# B&R Automation Studio project KeePak_Bliss_Reworked
Automation Studio 4.7.7.74 SP; technology packages: Acp10Arnc0 5.8.2, mapp 1.71.0, TextSystem 

## Configuration MasterConfiguration_ServoRam

CPU X20CP0484, AutomationRuntime C4.72, Build 4.1.2, Safety 1.10, Vc V4.72.0

### Task classes (Cpu.sw)
```
Cyclic#1 (cycle 4000 us, tolerance 0 us):
  ModeContro <- ModeControl.ModeControl_ST.prg
  GluePattCt <- Recipes.GluePattCtrl.prg
Cyclic#2 (cycle 8000 us, tolerance 8000 us):
  AdhesiveCo <- Actuators.AdhesiveControl.prg
  FoldPushCo <- Actuators.FoldPushControl.prg
  VacuumCont <- Actuators.VacuumControl.prg [disabled]
  ServoRamHa <- ServoMotion.ServoRamHandler.prg
  ServoFeedH <- ServoMotion.ServoFeedHandler.prg
  MotionHand <- ServoMotion.MotionHandler.prg
  MappCalls <- ServoMotion.MappCalls.prg
  ServoPnPHa <- ServoMotion.ServoPnPHandler.prg
  BodyHopper <- ServoMotion.BodyHopperHandler.prg
  LeftHopper <- ServoMotion.LeftHopperHandler.prg
  RightHoppe <- ServoMotion.RightHopperHandler.prg
Cyclic#3 (cycle 48000 us, tolerance 48000 us):
  SafetySamp <- AsSafetySolution.SafetySample.prg
Cyclic#4 (cycle 100000 us, tolerance 100000 us):
  FlexTest1 <- Actuators.FlexTest.prg
Cyclic#7 (cycle 20000 us, tolerance 30000000 us):
  AlarmHandl <- AlarmControl.AlarmHandling.prg
Cyclic#8 (cycle 8000 us, tolerance 30000000 us):
  Recipes <- Recipes.Recipes.prg
  HMIControl <- HMI.HMIControl.prg
  FlexTest <- Actuators.NordsonComm.NordsonMBComm.prg
  NordsonExt <- Actuators.NordsonComm.NordsonExtendedComm.prg
  PatliteCom <- Stacklight.PatliteComm.prg
DataObjects: assl1, Acp10sys
NcDataObjects: acp10etxen <- ServoMotion.acp10etxen.dob, gBHop <- gFeedobj.gBHop.dob, gFeedi <- gFeedobj.gFeedi.dob, brake <- gFeedobj.brake.dob, disablebra <- gFeedobj.disablebrakecheck.dob
VcDataObjects: Visu <- HMI.Visu.dob, Panel <- AsSafetySolution.Panel.dob
Binaries: vccbtn, vcpdvnc, arialbd, vcmgr, vctcal, vcgclass, vcfile, vcctext, vccnum, TCData, vcpkat, udbdef, vcfntttf, arial, vccshape, vcalarm, vccpwd, vcdsloc, Visu01, vccdt, vccscale, vcchspot, vccbmp, vccstr, vcshared, vcrt, vcnet, Visu02, calibri, vcbclass, vcdsint, vcpdsw, vccovl, Visu03, vccddbox, vccpopup, Panel03, Panel02, vcchtml, Panel01, vcxml, vccurl, arsvcreg, TCLang, vcpfgen, vcclbox, Acp10map, acp10cfg, ServoFeed, ServoRam, sysconf, AlarmCfg, RcpCfg, Role, User, ashwd, iomap, arconfig, AlrmHstCfg, TC, asfw, ashwac, ServoPnP, BodyHop, LeftHop, RightHop, ServoHop, vcpdi815, vcptelo, vcpdihd, vcpk, vcpfppc7, vcpdi855, vcpfar00, TopLinMot, BotLinMot, RamCfg
Libraries: operator, runtime, astime, AsIecCon, standard, brsystem, sys_lib, Constants, Vacuum, FoldPush, GluePatt, SetRamPars, GrayToBin, AsBrStr, InvErrTxt, DistCalc, AsSafety, FileIO, AsXml, AsMbTcp, asstring, AsIOAcc, AsBrMath, Lib_PBFlx, AsEPL, DataObj, AsIODiag, Acp10man, Acp10par, NcGlobal, Acp10sdc, Acp10sim, Acp10_MC, MpAxis, MpBase, MpAlarmX, MpCom, MpRecipe, MappCall, Types, AxisFUBs, vcresman, areventlog, powerlnk
```

### Hardware
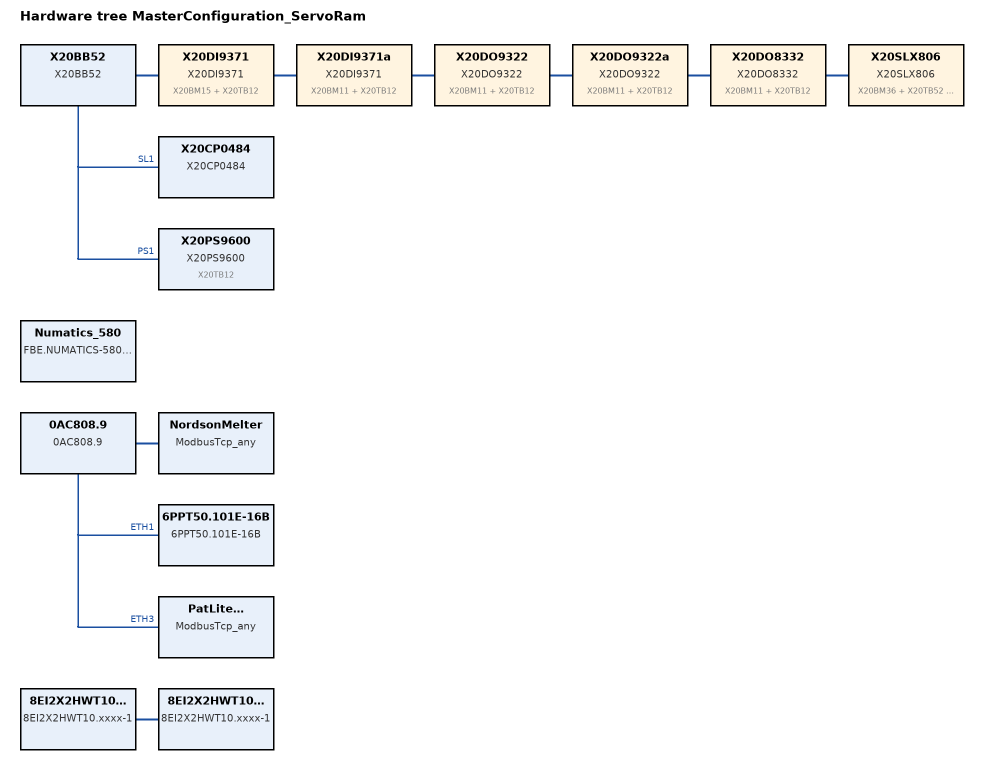
```
0AC808.9 : 0AC808.9 v1.0.0.0  [ETH1 -> 6PPT50.101E-16B.ETH1 [Cable Type=PowerlinkCable, Length=10, Version=1.0.0.2]; ETH2 -> NordsonMelter.ETH1 [Cable Type=PowerlinkCable, Length=10, Version=1.0.0.2]; ETH3 -> PatLite_LightStack.ETH1 [Cable Type=PowerlinkCable, Length=10, Version=1.0.0.2]]
6PPT50.101E-16B : 6PPT50.101E-16B v1.0.0.0  [ETH1 -> 0AC808.9.ETH1 [Cable Type=PowerlinkCable, Length=10, Version=1.0.0.2]; ETH2 -> X20CP0484.IF2 [Cable Type=PowerlinkCable, Length=10, Version=1.0.0.2]]
  Terminal = true
  Startmode = 1
  ShowBootlogoVNC = 1
  Mode = Manual
  InternetAddress = 192.168.0.222
  Subnetmask = 255.255.255.0
  ScreenRotation = 180
  SelectedFavoriteVNC = 192.168.0.100:5900
  Favorites_VNC1 = 192.168.0.100:5900  // Machine Display
  Favorites_VNC2 = 192.168.0.100:5901  // Safety Setup
  PasswordVNC = 2147
  LocalScaling = 1
  PasswordCIFS = 
  PasswordServiceEncrypt = 1
  PasswordServiceEncrypted = Sr1m/ubkTobKtMGmYG+OdX+pBVPXHNEV0toUjrnwIzvQUaZsN7HbgkMHcdX7NWbHkxunU2zcGZr9hHRCxdVEkcw0t0EkEZxQSM76MpE9s3WvBFtWwy/TiER4jA/5ccmygtG07vdCb9DlCJAeCcJdYe8VLadkZNOaNo2jGOliNnQ=
  VncKeyMappingFile = VC\6PPT30.101G-20B.dis
8EI2X2HWT10.xxxx-1 : 8EI2X2HWT10.xxxx-1 v2.2.0.1  [PLK2 -> 8EI2X2HWT10.xxxx-1a.PLK1 [Cable Type=PowerlinkCable, Length=10, Version=1.0.0.2]]
  MotionTP = Acp10Arnc0
  EnableDNA = on
  EPL_DNA_Head = 0
  EPL_DNA_Predecessor = 1
  Ax1Interface = Ax1EnDat
  Ax2Interface = Ax2EnDat
  Ax3Interface = Ax3EnDat
8EI2X2HWT10.xxxx-1a : 8EI2X2HWT10.xxxx-1 v2.2.0.1  [PLK1 -> 8EI2X2HWT10.xxxx-1.PLK2 [Cable Type=PowerlinkCable, Length=10, Version=1.0.0.2]; PLK2 -> X20CP0484.IF3 [Cable Type=PowerlinkCable, Length=10, Version=1.0.0.2]]
  MotionTP = Acp10Arnc0
  EnableDNA = on
  EPL_DNA_Head = 0
  EPL_DNA_HubPort = 1
  Ax1Interface = Ax1EnDat
  Ax2Interface = Ax2EnDat
  Ax3Interface = Ax3EnDat
NordsonMelter : ModbusTcp_any v1.0.6.0  [ETH1 -> 0AC808.9.ETH2 [Cable Type=PowerlinkCable, Length=10, Version=1.0.0.2]]
  IpAddress = 192.168.0.201
  UnitId = 1
Numatics_580 : FBE.NUMATICS-580-20150428-145500 v1.0 (OrderNumber=Numatics 580)
  Supervision = off
PatLite_LightStack : ModbusTcp_any v1.0.6.0 (Disabled=true)  [ETH1 -> 0AC808.9.ETH3 [Cable Type=PowerlinkCable, Length=10, Version=1.0.0.2]]
  Connector ETH2 (Disabled=true)
  IpAddress = 192.168.0.200
X20BB52 : X20BB52 v1.1.0.0
  Connector IF6:
    CycleTime = 2000
X20BM11 : X20BM11 v1.0.0.1  [X2X1 -> X20BM11b.X2X2]
X20BM11a : X20BM11 v1.0.0.1  [X2X1 -> X20BM15.X2X2]
X20BM11b : X20BM11 v1.0.0.1  [X2X1 -> X20BM11d.X2X2]
X20BM11d : X20BM11 v1.0.0.1  [X2X1 -> X20BM11a.X2X2]
X20BM15 : X20BM15 v1.0.1.0  [X2X1 -> X20BB52.IF6]
X20BM36 : X20BM36 v1.0.0.6  [X2X1 -> X20BM11.X2X2]
X20CP0484 : X20CP0484 v1.2.1.0  [SL -> X20BB52.SL1]
  Connector IF2:
    ActivateDevice = 1
    Mode = Manual
    InternetAddress = 192.168.0.100
    SubnetMask = 255.255.255.0
    InaNodeNumber = 0
    Vnc1
    VncVcObjectName1 = Visu
    VncKeyMappingFile1 = VC\PS2-Keyboard.dis
    VncAuthentication1 = 1
    VncPasswordViewOnly1 = 21472147
    VncPasswordViewControl1 = 2147
    VncMaxConnections1 = 4
    VncRefreshRate1 = 100
    Vnc2
    VncVcObjectName2 = Panel
    VncKeyMappingFile2 = VC\PS2-Keyboard1.dis
    VncAuthentication2 = 1
    VncPasswordViewOnly2 = 21472147
    VncPasswordViewControl2 = 2147
    VncPortNumber2 = 5901
    VncRefreshRate2 = 100
    ActivateModbus = 1
    NumSlaves = -1
    NumAllBlocks = -1
    MemSizeIn = -1
    MemSizeOut = -1
  Connector IF3:
    CycleTime = 4000
  ConfigurationID = KeePakVFDCaseErector_C70_10Inch
  UserPartitionSize = 100
  PermanentPvSize = 1024
  RemanentGlobalPvSize = 1024
  TimerDeviceType = EPLX2X
  TimerDevice = X20CP0484.IF3
  TaskClassIdleTime = 4000
  Cyclic1Duration = 4000
  Cyclic1Tolerance = 0
  Cyclic2Duration = 8000
  Cyclic2Tolerance = 8000
  Cyclic3Duration = 48000
  Cyclic3Tolerance = 48000
  Cyclic4Duration = 100000
  Cyclic4Tolerance = 100000
  Cyclic5Duration = 200000
  Cyclic5Tolerance = 200000
  Cyclic6Duration = 500000
  Cyclic6Tolerance = 500000
  Cyclic7Duration = 20000
  Cyclic7Tolerance = 30000000
  Cyclic8Duration = 8000
  Cyclic8Tolerance = 30000000
  FileDevice1
  FileDeviceName1 = recipes
  FileDevicePath1 = F:\
  EthernetDefaultGateway = 192.168.0.100
  FtpUser1
  FtpUsername1 = jeremy
  FtpUserPassword1 = CB9xa/tRkdxv0VtZFfoX4sbyc2/nOLcpzFFiUfDmX6w=
  FtpUserSalt1 = PVNzvqae
  FTPAccessRight1 = 0
X20DI9371 : X20DI9371 v1.0.2.0  [SS1 -> X20TB12.SS; SL -> X20BM15.SL1]
  Supervision = off
X20DI9371a : X20DI9371 v1.0.2.0  [SS1 -> X20TB12a.SS; SL -> X20BM11a.SL1]
X20DO8332 : X20DO8332 v1.0.2.0  [SS1 -> X20TB12e.SS; SL -> X20BM11.SL1]
  Supervision = off
  PowerSupply01 = on
X20DO9322 : X20DO9322 v1.0.3.0  [SS1 -> X20TB12d.SS; SL -> X20BM11d.SL1]
  Supervision = off
X20DO9322a : X20DO9322 v1.0.3.0  [SS1 -> X20TB12b.SS; SL -> X20BM11b.SL1]
X20PS9600 : X20PS9600 v1.0.1.0  [PS -> X20BB52.PS1; SS1 -> X20TB12f.SS]
X20SLX806 : X20SLX806 v1.10.5.0  [SS1 -> X20TB52.SS; SS2 -> X20TB52a.SS; SL -> X20BM36.SL1]
  Supervision = off
  SafeProject = SafeLOGIC-1
  SafeDesigner = 4.2.6.2
  DigitalOutput01 = viaSafeLOGIC
  DigitalOutput02 = viaSafeLOGIC
  DigitalOutput03 = viaSafeLOGIC
  DigitalOutput04 = viaSafeLOGIC
  DigitalOutput05 = viaSafeLOGIC
  DigitalOutput06 = viaSafeLOGIC
  UnsafeInputUINTs = 4
X20TB12 : X20TB12 v1.0.0.0
X20TB12a : X20TB12 v1.0.0.0
X20TB12b : X20TB12 v1.0.0.0
X20TB12d : X20TB12 v1.0.0.0
X20TB12e : X20TB12 v1.0.0.0
X20TB12f : X20TB12 v1.0.0.0
X20TB52 : X20TB52 v1.0.0.1
X20TB52a : X20TB52 v1.0.0.1
```

### Cpu.per - X20CP0484/Cpu.per
```iecst
VAR_CONFIG
	ServoFeed_EPD AT %M0; (* *)
	BodyHopper_EPD AT %M40; (* *)
	LeftHopper_EPD AT %M80; (* *)
	RightHopper_EPD AT %M120; (* *)
	ServoRam_EPD AT %M160; (* *)
	ServoPnP_EPD AT %M200; (* *)
	ServoRamFirstHomeExecuted AT %MX240; (* *)
	ServoFeedFirstHomeExecuted AT %MX241; (* *)
	BodyHopperFirstHomeExecuted AT %MX242; (* *)
	LeftHopperFirstHomeExecuted AT %MX243; (* *)
	RightHopperFirstHomeExecuted AT %MX244; (* *)
	ServoPnPFirstHomeExecuted AT %MX245; (* *)
	CycleCount AT %MD248; (* *)
	LubeCount AT %MD252; (* *)
END_VAR
```

### IoMap.iom - X20CP0484/IoMap.iom
```iecst
VAR_CONFIG
	Cyclic#1.::gIO.ModuleOKs[4] AT %IX."X20DO8332".ModuleOk;
	Cyclic#1.::gIO.DOs.GlueChannel1 AT %QX."X20DO8332".DigitalOutput01;
	Cyclic#1.::gIO.DOs.GlueChannel2 AT %QX."X20DO8332".DigitalOutput02;
	Cyclic#1.::gIO.DOs.GlueChannel3 AT %QX."X20DO8332".DigitalOutput03;
	Cyclic#1.::gIO.DOs.GlueChannel4 AT %QX."X20DO8332".DigitalOutput04;
	Cyclic#1.::gIO.DOs.ZeroEncoder AT %QX."X20DO8332".DigitalOutput08;
	Cyclic#1.::gIO.DOs.ResetSafety AT %QX."X20SLX806".BOOL101;
	Cyclic#1.::gIO.DIs.SafetyOK AT %IX."X20SLX806".BOOL001;
	Cyclic#1.::gIO.SafetyStatus.CabinetEStopStatus AT %IW."X20SLX806".UINT001;
	Cyclic#1.::gIO.SafetyStatus.SafetyProgramRunning AT %QX."X20SLX806".BOOL102;
	Cyclic#1.::gIO.SafetyStatus.SafetyProgramRunning AT %IX."X20SLX806".BOOL002;
	Cyclic#1.::gIO.ModuleOKs[6] AT %IX."X20SLX806".ModuleOk;
	Cyclic#1.::gIO.ModuleOKs[7] AT %IX."X20SC2212".ModuleOk;
	Cyclic#1.::gIO.SafetyStatus.GuardDoorsOK AT %IX."X20SLX806".BOOL003;
	Cyclic#1.::gIO.SafetyStatus.FrontEStopOK AT %IX."X20SLX806".BOOL004;
	Cyclic#1.::gIO.SafetyStatus.BackEstopOK AT %IX."X20SLX806".BOOL005;
	Cyclic#1.::gIO.DIs.AdhesivePhotoEye AT %IX."X20DI9371".DigitalInput01;
	Cyclic#1.::gIO.DIs.BodyDetect AT %IX."X20DI9371".DigitalInput04;
	Cyclic#1.::gIO.DIs.DownstreamSensorRaw AT %IX."X20DI9371".DigitalInput03;
	Cyclic#1.::gIO.DIs.BodyHopperLow AT %IX."X20DI9371".DigitalInput05;
	Cyclic#1.::gIO.DIs.AirPressureOK AT %IX."X20DI9371".DigitalInput02;
	::gIO.ModuleOKs[2] AT %IX."X20DI9371".ModuleOk;
	Cyclic#1.::gIO.DIs.BodyHopperMotor_OFF AT %IX."X20DI9371".DigitalInput09;
	Cyclic#1.::gIO.DIs.LeftHopperMotor_RUN AT %IX."X20DI9371".DigitalInput10;
	Cyclic#1.::gIO.DIs.LeftHopperMotor_OFF AT %IX."X20DI9371".DigitalInput11;
	Cyclic#1.::gIO.DIs.LeftHopperLow AT %IX."X20DI9371".DigitalInput06;
	Cyclic#1.::gIO.DIs.RightHopperLow AT %IX."X20DI9371".DigitalInput07;
	Cyclic#1.::gIO.DIs.BodyHopperMotor_RUN AT %IX."X20DI9371".DigitalInput08;
	Cyclic#1.::gIO.DIs.RightHopperMotor_RUN AT %IX."X20DI9371".DigitalInput12;
	Cyclic#1.::gIO.DOs.FoldingHoldVacuum AT %QX."X20DO9322".DigitalOutput03;
	Cyclic#1.::gIO.DOs.BodyVacuumOn AT %QX."X20DO9322".DigitalOutput01;
	Cyclic#1.::gIO.DOs.SidePanelHoldVacuum AT %QX."X20DO9322".DigitalOutput02;
	Cyclic#1.::gIO.DOs.PushOn AT %QX."X20DO9322".DigitalOutput04; (*24 VDC / 0.5 A, source **Normally the Pushers go here***)
	Cyclic#1.::gIO.DOs.AmberLightStack AT %QX."X20DO9322".DigitalOutput05;
	Cyclic#1.::gIO.DOs.GreenLightStack AT %QX."X20DO9322".DigitalOutput06;
	Cyclic#1.::gIO.DOs.RedLightStack AT %QX."X20DO9322".DigitalOutput07;
	Cyclic#1.::gIO.DOs.AirOn AT %QX."X20DO9322".DigitalOutput08;
	Cyclic#1.::gIO.DOs.Pneumatics580ControlWord1 AT %QW."Numatics_580".Out01_I3201Out;
	Cyclic#1.::gIO.ModuleOKs[7] AT %IX."Numatics_580".ModuleOk;
	Cyclic#1.::gIO.DIs.Pneumatics580StatusWord3 AT %IW."Numatics_580".In03_I3403;
	::b_ModuleStatus AT %IX."NordsonMelter".ModuleOk;
	Cyclic#1.::gIO.DIs.RightHopperMotor_OFF AT %IX."X20DI9371a".DigitalInput01;
	Cyclic#1.::gIO.DIs.BodyVacuumAchieved AT %IX."X20DI9371a".DigitalInput02;
	Cyclic#1.::gIO.DIs.SidePickVacuumAchieved AT %IX."X20DI9371a".DigitalInput03;
	Cyclic#1.::gIO.DIs.SideFoldVacuumAchieved AT %IX."X20DI9371a".DigitalInput04;
	Cyclic#1.::gIO.DOs.OutConveyorOn_1 AT %QX."X20DO9322".DigitalOutput09;
	Cyclic#1.::gIO.DOs.OutConveyorOn_2 AT %QX."X20DO9322".DigitalOutput10;
	Cyclic#1.::gIO.DOs.OutConveyorOn_3 AT %QX."X20DO9322".DigitalOutput11;
	Cyclic#1.::gIO.DOs.SidePickCylinder AT %QX."X20DO9322a".DigitalOutput01;
	Cyclic#1.::gIO.DOs.RightSideFoldCylinder AT %QX."X20DO9322a".DigitalOutput04;
	Cyclic#1.::gIO.DOs.LeftSideFoldCylinder AT %QX."X20DO9322a".DigitalOutput03;
	Cyclic#1.::gIO.DOs.CompressionCylinder AT %QX."X20DO9322a".DigitalOutput05;
	Cyclic#1.::gIO.DOs.BodyKicker AT %QX."X20DO9322".DigitalOutput12;
	Cyclic#1.::GuideCylinder AT %QX."X20DO9322a".DigitalOutput02;
	Cyclic#1.::gIO.DIs.LubricationCounter AT %IX."X20DI9371a".DigitalInput05;
	Cyclic#1.::gIO.DIs.BodyPickHome AT %IX."X20DI9371a".DigitalInput06;
END_VAR
```

### LeftHop.mpaxisbasic - X20CP0484/Motion/LeftHop.mpaxisbasic
```
Element mpLeftHopper (Type=mpaxisbasic)
  AxisConfiguration:
    Axis:
      MeasurementUnit = 1
  Alarms = MpAlarmX
    mapp.AlarmX.Core.Configuration:
      [0]:
        Severity = 110
      [1]:
        Severity = 110
      [2]:
        Severity = 110
      [3]:
        Severity = 110
      [4]:
        Severity = 110
      [5]:
        Severity = 110
      [6]:
        Severity = 110
      [7]:
        Severity = 110
      [8]:
        Severity = 110
      [9]:
        Severity = 110
      [10]:
        Severity = 110
      [11]:
        Severity = 110
      [12]:
        Severity = 110
      [13]:
        Severity = 110
      [14]:
        Severity = 110
      [15]:
        Severity = 110
```

- Safety project (password-protected, skipped)

## Logical view

### Global.var
```iecst
VAR RETAIN
	BodyHopperFirstHomeExecuted : BOOL;
	BodyHopper_EPD : MC_ENDLESS_POSITION;
END_VAR
VAR
	b_ModuleStatus : BOOL;
END_VAR
VAR RETAIN
	CycleCount : UDINT;
END_VAR
VAR
	DistanceAfterLatch : REAL;
	FeedInCycle : BOOL;
	FeedPosFinal : LREAL;
	FeedPositionCapture : LREAL;
	FeedServoBusy : BOOL;
	gActivePage : USINT;
	gAdhesiveCtrlInterface : AdhesiveCtrlInterface_typ;
	gAirPressureAlarmActive : BOOL;
	gAlarmActive : BOOL;
	gAlarmSystemActive : BOOL;
	gAutoTune : BOOL;
	gBodyHopper : ACP10AXIS_typ;
	gBodyHopperInterface : Axis_Interface_typ;
	gBotLinAxis : ACP10AXIS_typ;
	gBotLinAxis_1 : ACP10AXIS_typ;
	gChangePage : USINT;
	gCurrentLimitHit : BOOL;
	gCyclesToFinish : SINT;
	gDownstreamBlocked : BOOL;
END_VAR
VAR RETAIN
	gEndlessPosBot : MC_ENDLESS_POSITION;
	gEndlessPosTop : MC_ENDLESS_POSITION;
END_VAR
VAR
	gFoldPushCtrlInterface : FoldPushCtrlInterface_typ := (Parameters:=(LinMotBotFolder:=(Parameter:=(MpBasicParameters:=(Home:=(Mode:=mpAXIS_HOME_MODE_RESTORE_POS,Position:=0,StartVelocity:=25,HomingVelocity:=5,Acceleration:=500,StartDirection:=mpAXIS_HOME_DIR_NEGATIVE,TorqueLimit:=0.5,BlockDetectionPositionError:=4,PositionErrorStopLimit:=10),Jog:=(Velocity:=2)))),LinMotTopFolder:=(Parameter:=(MpBasicParameters:=(Home:=(Mode:=mpAXIS_HOME_MODE_RESTORE_POS,Position:=0,StartVelocity:=25,HomingVelocity:=5,Acceleration:=500,StartDirection:=mpAXIS_HOME_DIR_NEGATIVE,TorqueLimit:=0.5,BlockDetectionPositionError:=4,PositionErrorStopLimit:=10),Jog:=(Velocity:=2))))));
	gForceBodyKicker : BOOL;
	gHighSeverityAlarmActive : BOOL;
	gHMI : HMIControl_typ;
	gHomingParameters : Home_Parameters_typ;
	gIO : IO_typ;
	gIsSimulated : BOOL;
	gLeftHopper : ACP10AXIS_typ;
	gLeftHopperInterface : Axis_Interface_typ;
	gLowSeverityAlarmActive : BOOL;
	gModeControlInterface : ModeCtrlInterface_typ;
	gNumActiveAlarms : UDINT;
	gNumAlarms : UDINT;
	gOffDelayCompensation : REAL;
	gOnDelayCompensation : REAL;
END_VAR
VAR CONSTANT
	gPassword : ARRAY[0..2] OF STRING[80] := ['','0911','6866'];
END_VAR
VAR
	gPnPAtStopPosition : BOOL;
	gPusherOn : BOOL;
	gRamAtStopPosition : BOOL;
	gRamCtrlInterface : RamControlInterface_typ;
	gRamWaitingOnBox : BOOL;
END_VAR
VAR RETAIN
	gRecipeInterface : {REDUND_UNREPLICABLE} RecipeCtrlInterface_typ := (0);
END_VAR
VAR
	gRightHopper : ACP10AXIS_typ;
	gRightHopperInterface : Axis_Interface_typ;
	gSafetyNotOKAlarmActive : BOOL;
	gServoFeed : ACP10AXIS_typ;
	gServoFeedInterface : Axis_Interface_typ;
	gServoFeed_1 : ACP10AXIS_typ;
	gServoPnP : ACP10AXIS_typ;
	gServoPnPInterface : Axis_Interface_typ;
	gServoRam : ACP10AXIS_typ;
	gServoRamInterface : Axis_Interface_typ;
	gServoRam_1 : ACP10AXIS_typ;
	gSoftwareReset : BOOL;
	gTopLinAxis : ACP10AXIS_typ;
	gTopLinAxis_1 : ACP10AXIS_typ;
	GuideCylinder : BOOL;
	gUserLevel : USINT;
	gVacCtrlInterface : VacCtrlInterface_typ;
	HoperLowStop : BOOL;
	HopperLowTime : TIME := T#7s;
	InfeedBoxPresent : BOOL;
END_VAR
VAR RETAIN
	LeftHopperFirstHomeExecuted : BOOL;
	LeftHopper_EPD : MC_ENDLESS_POSITION;
	LubeCount : UDINT;
END_VAR
VAR
	LubricationOK : BOOL;
	Melter : DUT_NDSN_Flex;
	PhotoEyeSeen : BOOL;
END_VAR
VAR RETAIN
	RightHopperFirstHomeExecuted : BOOL;
	RightHopper_EPD : MC_ENDLESS_POSITION;
	ServoFeedFirstHomeExecuted : BOOL;
	ServoFeed_EPD : MC_ENDLESS_POSITION;
END_VAR
VAR
	ServoPnPAutoHome : BOOL;
END_VAR
VAR RETAIN
	ServoPnPFirstHomeExecuted : BOOL;
	ServoPnP_EPD : MC_ENDLESS_POSITION;
END_VAR
VAR
	ServoRamAutoHome : BOOL;
	ServoRamBusy : BOOL;
	ServoRamClear : BOOL;
END_VAR
VAR RETAIN
	ServoRamFirstHomeExecuted : BOOL;
END_VAR
VAR
	ServoRamTrigger : BOOL;
END_VAR
VAR RETAIN
	ServoRam_EPD : MC_ENDLESS_POSITION;
END_VAR
VAR
	StopFeed : BOOL;
END_VAR
```

### Program Logical/Actuators/AdhesiveControl

#### Init.st
```iecst
PROGRAM _INIT
	(* Insert code here *)
	gAdhesiveCtrlInterface.Parameters.NumAdhesiveChannels := 4;

	DistanceAfterLatch := 1500; //make this large so that the machine doesn't start dispensing glue before it ever sees a photo eye. This will reset to 0 and count up once the photo eye is seen

END_PROGRAM
```

### Program Logical/Actuators/NordsonComm/NordsonMBComm

#### MbApp.typ
```iecst
(********************************************************************
 * COPYRIGHT -- Bernecker + Rainer
 ********************************************************************
 * Program: MbApp
 * File: MbApp.typ
 * Author: Bernecker + Rainer
 * Created: October 22, 2009
 ********************************************************************
 * Local data types of program MbApp
 ********************************************************************)

TYPE
	ModbusTCP_Handling_States_enum :
		(
		MB_IDLE := 0,
		MB_REQUEST_SET_TEMPS2,
		MB_REQUEST_SET_TEMPS,
		MB_READ_SET_TEMPS2,
		MB_READ_SET_TEMPS,
		MB_REQUEST_ACT_TEMPS2,
		MB_REQUEST_ACT_TEMPS,
		MB_READ_ACT_TEMPS2,
		MB_READ_ACT_TEMPS,
		MB_REQUEST_MELTER_STATUS,
		MB_READ_MELTER_STATUS,
		MB_REQUEST_ADH_USE,
		MB_READ_ADH_USE,
		MB_WRITE_REGISTERS,
		MB_READ_REGISTERS,
		MB_REQUEST_MACHINE_STATUS,
		MB_WRITE_SET_TEMP2,
		MB_WRITE_SET_TEMP,
		MB_VERIFY_SET_TEMP_WRITE2,
		MB_VERIFY_SET_TEMP_WRITE,
		MB_REQUEST_ATS_ALARMS,
		MB_READ_ATS_ALARMS,
		MB_ERROR := 999
		);
END_TYPE
```

#### MbApp.var
```iecst
(********************************************************************
 * COPYRIGHT -- Bernecker + Rainer
 ********************************************************************
 * Program: MbApp
 * File: MbApp.var
 * Author: Bernecker + Rainer
 * Created: October 22, 2009
 ********************************************************************
 * Local variables of program MbApp
 ********************************************************************)
VAR
	state : ModbusTCP_Handling_States_enum;
	mb_station : STRING[50];
	write_register_address : UINT;
	num_registers_to_write : UINT;
	read_register_address : UINT;
	num_registers_to_read : UINT;
	ReadMultipleRegisters : mbReadHoldingRegisters;
	WriteMultipleRegisters : mbWriteMultipleRegisters;
	MBError : UINT;
	testIdx : USINT;
	DummyPacket2 : NordsonRxPacket_typ;
	DummyPacket : NordsonRxPacket_typ;
	NordsonRxPacket : NordsonRxPacket_typ;
	testChannel : USINT;
	NordsonTxPacket : NordsonTxPacket_typ;
	FeedbackCycleTimer : TON;
	MelterCmd : USINT;
	TempChannelToWrite : USINT;
	StandbyTimer : TON;
	FirstTimeCopySetTemps : BOOL;
END_VAR
```

#### MbApp.st
```iecst
(********************************************************************
 * COPYRIGHT -- Bernecker + Rainer
 ********************************************************************
 * Program: MbApp
 * File: MbApp.st
 * Author: Bernecker + Rainer
 * Created: October 22, 2009
 ********************************************************************
 * Implementation of program MbApp
 * State Nomenclature: "request" is a write to the nordson melter asking for some data
 * 					   "read" is a read from the nordson melter of the previously requested data
 *                     "write" is a write to the nordson melter asking to write some data to the melter
 *                     "verify" is a read from the nordson melter where we check to see that the write was accepted
 ********************************************************************)

PROGRAM _INIT

	NordsonTxPacket.Byte0_MelterControl := 16#1;
	NordsonTxPacket.Byte1_Command := 3;
	NordsonTxPacket.Byte2_Data_Index := 16#78;
	NordsonTxPacket.Byte3_Channel_Num := 16#3;
	NordsonTxPacket.Byte4_5_WriteData := 0;
	NordsonTxPacket.Byte6_7_Mot1Spd := 0;
	NordsonTxPacket.Byte8_9_Mot2Spd := 0;
	NordsonTxPacket.Byte10_11_Mot3Spd := 0;
	NordsonTxPacket.Byte12_13_Mot4Spd := 0;
	NordsonTxPacket.Byte14_15_NotUsed := 0;

	state := MB_IDLE;

	(* init values *)
	mb_station 			:= 'IF2.ST2';					(* path to modbus station *)
	write_register_address	:= 1024;						(* register address on modbus station *)
	read_register_address	:= 0;						(* register address on modbus station *)
	num_registers_to_write := 8;
	num_registers_to_read := 8;

	testChannel := CHANNEL_ACT_TEMP_START;
	testIdx := IDX_ACT_TEMP;

	gAdhesiveCtrlInterface.Commands.MelterOn := TRUE;
	gAdhesiveCtrlInterface.Commands.PumpsOn := TRUE;
	//gAdhesiveCtrlInterface.Parameters.NordsonComms.StandbyTimeoutTime := T#2h;
	//Removed Standby due to Waco machine going into Standby at random times. Added 05/15/2024

	FirstTimeCopySetTemps := FALSE;

END_PROGRAM

PROGRAM _CYCLIC

	IF(gAdhesiveCtrlInterface.Parameters.FeedbackIsModbusTCP) THEN
		gHMI.StatusDatapoints.NordsonModbusSDP := UNHIDE + UNLOCK;
	ELSE
		gHMI.StatusDatapoints.NordsonModbusSDP := HIDE + LOCK;
	END_IF

	//StandbyTimer.IN := NOT(gRamCtrlInterface.Status.Running) AND NOT(gAdhesiveCtrlInterface.Commands.MelterStandbyOn);
	StandbyTimer.IN := NOT(gServoRamInterface.Status.InMotion OR gServoPnPInterface.Status.InMotion OR gServoFeedInterface.Status.InMotion OR
							gBodyHopperInterface.Status.InMotion OR gLeftHopperInterface.Status.InMotion OR gRightHopperInterface.Status.InMotion)
						AND NOT(gAdhesiveCtrlInterface.Commands.MelterStandbyOn);

	StandbyTimer.PT := gAdhesiveCtrlInterface.Parameters.NordsonComms.StandbyTimeoutTime;
	StandbyTimer();

	IF(StandbyTimer.Q) THEN
		gAdhesiveCtrlInterface.Commands.MelterStandbyOn := TRUE;
	END_IF

	//clearing standby on command shiuld turn standby off. Changed standbyoff to True
	IF(gAdhesiveCtrlInterface.Commands.MelterStandbyOff) THEN
		gAdhesiveCtrlInterface.Commands.MelterStandbyOff := TRUE;
		gAdhesiveCtrlInterface.Commands.MelterStandbyOn := FALSE;
	END_IF

	IF((gAdhesiveCtrlInterface.Status.NordsonInStandby) AND (gAdhesiveCtrlInterface.Parameters.FeedbackIsModbusTCP)) THEN
		gHMI.StatusDatapoints.NordsonStandbyOffSDP := UNHIDE + UNLOCK;
	ELSE
		gHMI.StatusDatapoints.NordsonStandbyOffSDP := HIDE + LOCK;
	END_IF

	//if nordson feedback is bypassed, the error count should reset to 0
	IF gAdhesiveCtrlInterface.Parameters.NordsonComms.ByPassFeedback THEN
		gAdhesiveCtrlInterface.Parameters.NordsonComms.ConsecutiveErrorCount := 0;
	END_IF

	CASE state OF

		MB_IDLE:
			FeedbackCycleTimer.IN := ((gAdhesiveCtrlInterface.Parameters.FeedbackIsModbusTCP) AND (gAdhesiveCtrlInterface.Parameters.NordsonComms.ByPassFeedback = FALSE));

			IF(gAdhesiveCtrlInterface.Parameters.FeedbackIsModbusTCP = FALSE) THEN
				gAdhesiveCtrlInterface.Parameters.NordsonComms.ConsecutiveErrorCount := 0;
			END_IF

			IF(gAdhesiveCtrlInterface.Commands.WriteChannelTemp) THEN
				gAdhesiveCtrlInterface.Commands.WriteChannelTemp := FALSE;
				IF gAdhesiveCtrlInterface.Parameters.NordsonComms.GlobalSetTemp <> 0 THEN
					gAdhesiveCtrlInterface.Parameters.NordsonComms.ChannelSetTempRequested[0] := gAdhesiveCtrlInterface.Parameters.NordsonComms.GlobalSetTemp;
					gAdhesiveCtrlInterface.Parameters.NordsonComms.ChannelSetTempRequested[1] := gAdhesiveCtrlInterface.Parameters.NordsonComms.GlobalSetTemp;
					gAdhesiveCtrlInterface.Parameters.NordsonComms.ChannelSetTempRequested[2] := gAdhesiveCtrlInterface.Parameters.NordsonComms.GlobalSetTemp;
					gAdhesiveCtrlInterface.Parameters.NordsonComms.ChannelSetTempRequested[3] := gAdhesiveCtrlInterface.Parameters.NordsonComms.GlobalSetTemp;
					gAdhesiveCtrlInterface.Parameters.NordsonComms.ChannelSetTempRequested[4] := gAdhesiveCtrlInterface.Parameters.NordsonComms.GlobalSetTemp;
					gAdhesiveCtrlInterface.Parameters.NordsonComms.ChannelSetTempRequested[5] := gAdhesiveCtrlInterface.Parameters.NordsonComms.GlobalSetTemp;
					gAdhesiveCtrlInterface.Parameters.NordsonComms.ChannelSetTempRequested[6] := gAdhesiveCtrlInterface.Parameters.NordsonComms.GlobalSetTemp;
					gAdhesiveCtrlInterface.Parameters.NordsonComms.ChannelSetTempRequested[7] := gAdhesiveCtrlInterface.Parameters.NordsonComms.GlobalSetTemp;
					gAdhesiveCtrlInterface.Parameters.NordsonComms.ChannelSetTempRequested[8] := gAdhesiveCtrlInterface.Parameters.NordsonComms.GlobalSetTemp;
					gAdhesiveCtrlInterface.Parameters.NordsonComms.ChannelSetTempRequested[9] := gAdhesiveCtrlInterface.Parameters.NordsonComms.GlobalSetTemp;
					gAdhesiveCtrlInterface.Parameters.NordsonComms.GlobalSetTemp := 0;
				END_IF
				TempChannelToWrite := 0;
				state := MB_WRITE_SET_TEMP;

			ELSIF(FeedbackCycleTimer.Q) THEN
				FeedbackCycleTimer.IN := FALSE;
				state := MB_REQUEST_MELTER_STATUS;
			END_IF

		MB_REQUEST_MELTER_STATUS:

			WriteMultipleRegisters.enable := 1;
			NordsonTxPacket.Byte0_MelterControl := MelterCmd;
			NordsonTxPacket.Byte1_Command := READ_COMMAND;
			NordsonTxPacket.Byte2_Data_Index := IDX_MELTER_STATUS;
			NordsonTxPacket.Byte3_Channel_Num := 0;

			IF((WriteMultipleRegisters.status = ERR_FUB_ENABLE_FALSE) OR (WriteMultipleRegisters.status = ERR_FUB_BUSY)) THEN
				//do nothing
			ELSIF(WriteMultipleRegisters.status = ERR_OK) THEN
				WriteMultipleRegisters.enable := 0;
				state := MB_READ_MELTER_STATUS;
			ELSE
				WriteMultipleRegisters.enable := 0;
				MBError := WriteMultipleRegisters.status;
				state := MB_ERROR;
			END_IF

		MB_READ_MELTER_STATUS:

			ReadMultipleRegisters.enable := 1;

			IF((ReadMultipleRegisters.status = ERR_FUB_ENABLE_FALSE) OR (ReadMultipleRegisters.status = ERR_FUB_BUSY)) THEN
				//do nothing
			ELSIF(ReadMultipleRegisters.status = ERR_OK) THEN

				ReadMultipleRegisters.enable := 0;

				IF(NordsonRxPacket.Byte2_Ack_Data_Index = NordsonTxPacket.Byte2_Data_Index) THEN

					gAdhesiveCtrlInterface.Parameters.NordsonComms.MelterStatus := NordsonRxPacket.Byte4_5_Read_Data_0;
					gAdhesiveCtrlInterface.Parameters.NordsonComms.MelterIsOn := (gAdhesiveCtrlInterface.Parameters.NordsonComms.MelterStatus <> 8); //melter status == 8 => melter is not on

					DecodeStatus;

					//the melter MUST see a 0 for its ON command before it sees a 1. Send a 0 if the unit is faulted OR we have previously told it to turn on. and it never came on
				//	IF((gAdhesiveCtrlInterface.Parameters.NordsonComms.UnitFaulted) OR ((gAdhesiveCtrlInterface.Parameters.NordsonComms.MelterIsOn = FALSE) AND (NordsonTxPacket.Byte0_MelterControl.0 = TRUE))) THEN
					IF((gAdhesiveCtrlInterface.Parameters.NordsonComms.MelterIsOn = FALSE) AND (NordsonTxPacket.Byte0_MelterControl.0 = TRUE)) THEN
						MelterCmd := MELTER_OFF + PUMPS_OFF; //melter off, pumps off
					ELSE

						MelterCmd := 0;
						IF(gAdhesiveCtrlInterface.Commands.MelterOn) THEN
							MelterCmd := MelterCmd + MELTER_ON;
						END_IF

						IF((gAdhesiveCtrlInterface.Commands.PumpsOn) AND (gAdhesiveCtrlInterface.Status.UnitReady)) THEN
							MelterCmd := MelterCmd + PUMPS_ON; //only turn the pump on if the melter is ready
						END_IF

						IF((gAdhesiveCtrlInterface.Commands.MelterStandbyOn = FALSE) OR ((gAdhesiveCtrlInterface.Status.NordsonInStandby = FALSE) AND NordsonTxPacket.Byte0_MelterControl.6 = TRUE)) THEN
							//do not standby on
						ELSIF (gAdhesiveCtrlInterface.Commands.MelterStandbyOn = TRUE) THEN
							MelterCmd := MelterCmd + STANDBY_ON; //only turn the pump on if the melter is ready
						END_IF
					END_IF

					state := MB_REQUEST_SET_TEMPS;
				ELSE
					//stay in this state and re-execute read
				END_IF

			ELSE
				ReadMultipleRegisters.enable := 0;
				MBError := ReadMultipleRegisters.status;
				state := MB_ERROR;
			END_IF

		MB_REQUEST_SET_TEMPS:

			WriteMultipleRegisters.enable := 1;
			NordsonTxPacket.Byte0_MelterControl := MelterCmd;
			NordsonTxPacket.Byte1_Command := READ_COMMAND;
			NordsonTxPacket.Byte2_Data_Index := IDX_SET_TEMP;
			NordsonTxPacket.Byte3_Channel_Num := CHANNEL_SET_TEMP_START;

			IF((WriteMultipleRegisters.status = ERR_FUB_ENABLE_FALSE) OR (WriteMultipleRegisters.status = ERR_FUB_BUSY)) THEN
				//do nothing
			ELSIF(WriteMultipleRegisters.status = ERR_OK) THEN
				WriteMultipleRegisters.enable := 0;
				gAdhesiveCtrlInterface.Parameters.NordsonComms.ConsecutiveErrorCount := 0;
				state := MB_READ_SET_TEMPS;
			ELSE
				WriteMultipleRegisters.enable := 0;
				MBError := WriteMultipleRegisters.status;
				state := MB_ERROR;
			END_IF

		MB_READ_SET_TEMPS:

			ReadMultipleRegisters.enable := 1;

			IF((ReadMultipleRegisters.status = ERR_FUB_ENABLE_FALSE) OR (ReadMultipleRegisters.status = ERR_FUB_BUSY)) THEN
				//do nothing
			ELSIF(ReadMultipleRegisters.status = ERR_OK) THEN
				ReadMultipleRegisters.enable := 0;
				gAdhesiveCtrlInterface.Parameters.NordsonComms.ConsecutiveErrorCount := 0;

				IF((NordsonRxPacket.Byte2_Ack_Data_Index = NordsonTxPacket.Byte2_Data_Index) AND
					(NordsonRxPacket.Byte3_Ack_Channel_Num = NordsonTxPacket.Byte3_Channel_Num)) THEN

					DecodeStatus;

					gAdhesiveCtrlInterface.Parameters.NordsonComms.ChannelSetTempActual[0] := NordsonRxPacket.Byte4_5_Read_Data_0;
					gAdhesiveCtrlInterface.Parameters.NordsonComms.ChannelSetTempActual[1] := NordsonRxPacket.Byte6_7_Read_Data_1;
					gAdhesiveCtrlInterface.Parameters.NordsonComms.ChannelSetTempActual[2] := NordsonRxPacket.Byte8_9_Read_Data_2;
					gAdhesiveCtrlInterface.Parameters.NordsonComms.ChannelSetTempActual[3] := NordsonRxPacket.Byte10_11_Read_Data_3;
					gAdhesiveCtrlInterface.Parameters.NordsonComms.ChannelSetTempActual[4] := NordsonRxPacket.Byte12_13_Read_Data_4;
                    gAdhesiveCtrlInterface.Parameters.NordsonComms.ChannelSetTempActual[5] := NordsonRxPacket.Byte14_15_Read_Data_5;

					IF (FirstTimeCopySetTemps = FALSE) THEN
						gAdhesiveCtrlInterface.Parameters.NordsonComms.ChannelSetTempRequested := gAdhesiveCtrlInterface.Parameters.NordsonComms.ChannelSetTempActual;
						FirstTimeCopySetTemps := TRUE;
					END_IF

					state := MB_REQUEST_SET_TEMPS2; //for now, just go back to idle. Future versions need to read more stuff
				ELSE
					//stay in this state and re-execute read
				END_IF
			ELSE
				ReadMultipleRegisters.enable := 0;
				MBError := ReadMultipleRegisters.status;
				state := MB_ERROR;
			END_IF

		MB_REQUEST_SET_TEMPS2:

			WriteMultipleRegisters.enable := 1;
			NordsonTxPacket.Byte0_MelterControl := MelterCmd;
			NordsonTxPacket.Byte1_Command := READ_COMMAND;
			NordsonTxPacket.Byte2_Data_Index := IDX_SET_TEMP;
			NordsonTxPacket.Byte3_Channel_Num := 7;

			IF((WriteMultipleRegisters.status = ERR_FUB_ENABLE_FALSE) OR (WriteMultipleRegisters.status = ERR_FUB_BUSY)) THEN
				//do nothing
			ELSIF(WriteMultipleRegisters.status = ERR_OK) THEN
				WriteMultipleRegisters.enable := 0;
				gAdhesiveCtrlInterface.Parameters.NordsonComms.ConsecutiveErrorCount := 0;
				state := MB_READ_SET_TEMPS2;
			ELSE
				WriteMultipleRegisters.enable := 0;
				MBError := WriteMultipleRegisters.status;
				state := MB_ERROR;
			END_IF

		MB_READ_SET_TEMPS2:

			ReadMultipleRegisters.enable := 1;

			IF((ReadMultipleRegisters.status = ERR_FUB_ENABLE_FALSE) OR (ReadMultipleRegisters.status = ERR_FUB_BUSY)) THEN
				//do nothing
			ELSIF(ReadMultipleRegisters.status = ERR_OK) THEN
				ReadMultipleRegisters.enable := 0;
				gAdhesiveCtrlInterface.Parameters.NordsonComms.ConsecutiveErrorCount := 0;

				IF((NordsonRxPacket.Byte2_Ack_Data_Index = NordsonTxPacket.Byte2_Data_Index) AND
					(NordsonRxPacket.Byte3_Ack_Channel_Num = NordsonTxPacket.Byte3_Channel_Num)) THEN

					DecodeStatus;

					gAdhesiveCtrlInterface.Parameters.NordsonComms.ChannelSetTempActual[6] := NordsonRxPacket.Byte4_5_Read_Data_0;
					gAdhesiveCtrlInterface.Parameters.NordsonComms.ChannelSetTempActual[7] := NordsonRxPacket.Byte6_7_Read_Data_1;
					gAdhesiveCtrlInterface.Parameters.NordsonComms.ChannelSetTempActual[8] := NordsonRxPacket.Byte8_9_Read_Data_2;
					gAdhesiveCtrlInterface.Parameters.NordsonComms.ChannelSetTempActual[9] := NordsonRxPacket.Byte10_11_Read_Data_3;

					IF (FirstTimeCopySetTemps = FALSE) THEN
						gAdhesiveCtrlInterface.Parameters.NordsonComms.ChannelSetTempRequested := gAdhesiveCtrlInterface.Parameters.NordsonComms.ChannelSetTempActual;
						FirstTimeCopySetTemps := TRUE;
					END_IF

					state := MB_REQUEST_ACT_TEMPS; //for now, just go back to idle. Future versions need to read more stuff
				ELSE
					//stay in this state and re-execute read
				END_IF
			ELSE
				ReadMultipleRegisters.enable := 0;
				MBError := ReadMultipleRegisters.status;
				state := MB_ERROR;
			END_IF

		MB_REQUEST_ACT_TEMPS:

			WriteMultipleRegisters.enable := 1;
			NordsonTxPacket.Byte0_MelterControl := MelterCmd;
			NordsonTxPacket.Byte1_Command := READ_COMMAND;
			NordsonTxPacket.Byte2_Data_Index := IDX_ACT_TEMP;
			NordsonTxPacket.Byte3_Channel_Num := CHANNEL_ACT_TEMP_START;

			IF((WriteMultipleRegisters.status = ERR_FUB_ENABLE_FALSE) OR (WriteMultipleRegisters.status = ERR_FUB_BUSY)) THEN
				//do nothing
			ELSIF(WriteMultipleRegisters.status = ERR_OK) THEN
				WriteMultipleRegisters.enable := 0;
				state := MB_READ_ACT_TEMPS;
			ELSE
				WriteMultipleRegisters.enable := 0;
				MBError := WriteMultipleRegisters.status;
				state := MB_ERROR;
			END_IF

		MB_READ_ACT_TEMPS:

			ReadMultipleRegisters.enable := 1;

			IF((ReadMultipleRegisters.status = ERR_FUB_ENABLE_FALSE) OR (ReadMultipleRegisters.status = ERR_FUB_BUSY)) THEN
				//do nothing
			ELSIF(ReadMultipleRegisters.status = ERR_OK) THEN
				ReadMultipleRegisters.enable := 0;

				IF((NordsonRxPacket.Byte2_Ack_Data_Index = NordsonTxPacket.Byte2_Data_Index) AND
					(NordsonRxPacket.Byte3_Ack_Channel_Num = NordsonTxPacket.Byte3_Channel_Num)) THEN

					DecodeStatus;

					DummyPacket := NordsonRxPacket;

					gAdhesiveCtrlInterface.Parameters.NordsonComms.ChannelActTemp[0] := NordsonRxPacket.Byte4_5_Read_Data_0;
					gAdhesiveCtrlInterface.Parameters.NordsonComms.ChannelActTemp[1] := NordsonRxPacket.Byte6_7_Read_Data_1;
					gAdhesiveCtrlInterface.Parameters.NordsonComms.ChannelActTemp[2] := NordsonRxPacket.Byte8_9_Read_Data_2;
					gAdhesiveCtrlInterface.Parameters.NordsonComms.ChannelActTemp[3] := NordsonRxPacket.Byte10_11_Read_Data_3;
					gAdhesiveCtrlInterface.Parameters.NordsonComms.ChannelActTemp[4] := NordsonRxPacket.Byte12_13_Read_Data_4;
                    gAdhesiveCtrlInterface.Parameters.NordsonComms.ChannelActTemp[5] := NordsonRxPacket.Byte14_15_Read_Data_5;

					state := MB_REQUEST_ACT_TEMPS2;
				ELSE
					//stay in this state and re-execute read
				END_IF

			ELSE
				ReadMultipleRegisters.enable := 0;
				MBError := ReadMultipleRegisters.status;
				state := MB_ERROR;
			END_IF

		MB_REQUEST_ACT_TEMPS2:

			WriteMultipleRegisters.enable := 1;
			NordsonTxPacket.Byte0_MelterControl := MelterCmd;
			NordsonTxPacket.Byte1_Command := READ_COMMAND;
			NordsonTxPacket.Byte2_Data_Index := IDX_ACT_TEMP;
			NordsonTxPacket.Byte3_Channel_Num := 7;

			IF((WriteMultipleRegisters.status = ERR_FUB_ENABLE_FALSE) OR (WriteMultipleRegisters.status = ERR_FUB_BUSY)) THEN
				//do nothing
			ELSIF(WriteMultipleRegisters.status = ERR_OK) THEN
				WriteMultipleRegisters.enable := 0;
				state := MB_READ_ACT_TEMPS2;
			ELSE
				WriteMultipleRegisters.enable := 0;
				MBError := WriteMultipleRegisters.status;
				state := MB_ERROR;
			END_IF

		MB_READ_ACT_TEMPS2:

			ReadMultipleRegisters.enable := 1;

			IF((ReadMultipleRegisters.status = ERR_FUB_ENABLE_FALSE) OR (ReadMultipleRegisters.status = ERR_FUB_BUSY)) THEN
				//do nothing
			ELSIF(ReadMultipleRegisters.status = ERR_OK) THEN
				ReadMultipleRegisters.enable := 0;

				IF((NordsonRxPacket.Byte2_Ack_Data_Index = NordsonTxPacket.Byte2_Data_Index) AND
					(NordsonRxPacket.Byte3_Ack_Channel_Num = NordsonTxPacket.Byte3_Channel_Num)) THEN

					DecodeStatus;

					DummyPacket2 := NordsonRxPacket;

					gAdhesiveCtrlInterface.Parameters.NordsonComms.ChannelActTemp[6] := NordsonRxPacket.Byte4_5_Read_Data_0;
					gAdhesiveCtrlInterface.Parameters.NordsonComms.ChannelActTemp[7] := NordsonRxPacket.Byte6_7_Read_Data_1;
					gAdhesiveCtrlInterface.Parameters.NordsonComms.ChannelActTemp[8] := NordsonRxPacket.Byte8_9_Read_Data_2;
					gAdhesiveCtrlInterface.Parameters.NordsonComms.ChannelActTemp[9] := NordsonRxPacket.Byte10_11_Read_Data_3;

					state := MB_REQUEST_ATS_ALARMS;
				ELSE
					//stay in this state and re-execute read
				END_IF

			ELSE
				ReadMultipleRegisters.enable := 0;
				MBError := ReadMultipleRegisters.status;
				state := MB_ERROR;
			END_IF

		MB_REQUEST_ATS_ALARMS:

			WriteMultipleRegisters.enable := 1;
			NordsonTxPacket.Byte0_MelterControl := MelterCmd;
			NordsonTxPacket.Byte1_Command := READ_COMMAND;
			NordsonTxPacket.Byte2_Data_Index := IDX_ATS_ALARMS;

			IF((WriteMultipleRegisters.status = ERR_FUB_ENABLE_FALSE) OR (WriteMultipleRegisters.status = ERR_FUB_BUSY)) THEN
				//do nothing
			ELSIF(WriteMultipleRegisters.status = ERR_OK) THEN
				WriteMultipleRegisters.enable := 0;
				state := MB_READ_ATS_ALARMS;
			ELSE
				WriteMultipleRegisters.enable := 0;
				MBError := WriteMultipleRegisters.status;
				state := MB_ERROR;
			END_IF

		MB_READ_ATS_ALARMS:

			ReadMultipleRegisters.enable := 1;

			IF((ReadMultipleRegisters.status = ERR_FUB_ENABLE_FALSE) OR (ReadMultipleRegisters.status = ERR_FUB_BUSY)) THEN
				//do nothing
			ELSIF(ReadMultipleRegisters.status = ERR_OK) THEN
				ReadMultipleRegisters.enable := 0;

				IF(NordsonRxPacket.Byte2_Ack_Data_Index = NordsonTxPacket.Byte2_Data_Index) THEN

					DecodeStatus;

					gAdhesiveCtrlInterface.Status.ATS_AddOnOverLimit := NordsonRxPacket.Byte4_5_Read_Data_0.0;
					gAdhesiveCtrlInterface.Status.ATS_AddOnUnderLimit := NordsonRxPacket.Byte4_5_Read_Data_0.1;

					state := MB_IDLE;
				ELSE
					//stay in this state and re-execute read
				END_IF

			ELSE
				ReadMultipleRegisters.enable := 0;
				MBError := ReadMultipleRegisters.status;
				state := MB_ERROR;
			END_IF

		MB_WRITE_SET_TEMP:

			WriteMultipleRegisters.enable := 1;
			NordsonTxPacket.Byte0_MelterControl := MelterCmd;
			NordsonTxPacket.Byte1_Command := WRITE_COMMAND;
			NordsonTxPacket.Byte2_Data_Index := IDX_SET_TEMP;
			NordsonTxPacket.Byte3_Channel_Num := TempChannelToWrite + 1; //TempChannelToWrite starts counting at 0, but nordson melter starts counting at 1
			NordsonTxPacket.Byte4_5_WriteData := gAdhesiveCtrlInterface.Parameters.NordsonComms.ChannelSetTempRequested[TempChannelToWrite];

			IF((WriteMultipleRegisters.status = ERR_FUB_ENABLE_FALSE) OR (WriteMultipleRegisters.status = ERR_FUB_BUSY)) THEN
				//do nothing
			ELSIF(WriteMultipleRegisters.status = ERR_OK) THEN
				WriteMultipleRegisters.enable := 0;
				state := MB_VERIFY_SET_TEMP_WRITE;
			ELSE
				WriteMultipleRegisters.enable := 0;
				MBError := WriteMultipleRegisters.status;
				state := MB_ERROR;
			END_IF

		MB_VERIFY_SET_TEMP_WRITE:

			ReadMultipleRegisters.enable := 1;

			IF((ReadMultipleRegisters.status = ERR_FUB_ENABLE_FALSE) OR (ReadMultipleRegisters.status = ERR_FUB_BUSY)) THEN
				//do nothing
			ELSIF(ReadMultipleRegisters.status = ERR_OK) THEN
				ReadMultipleRegisters.enable := 0;

				IF((NordsonRxPacket.Byte2_Ack_Data_Index = NordsonTxPacket.Byte2_Data_Index) AND
					(NordsonRxPacket.Byte3_Ack_Channel_Num = NordsonTxPacket.Byte3_Channel_Num)) THEN

					DecodeStatus;

					IF(TempChannelToWrite < NUM_NORDSON_TEMP_ZONES_M1) THEN
						IF(TempChannelToWrite = 0) THEN
							TempChannelToWrite := 2; //channel 0 and 1 get the same temp, no need to re-write channel 1
							state := MB_WRITE_SET_TEMP;
						ELSE
							TempChannelToWrite := TempChannelToWrite + 1; //set the temperature for the next channel (Skip channel 2). Machine has 3 total channels
							state := MB_WRITE_SET_TEMP;
						END_IF
					ELSE
						state := MB_IDLE;
					END_IF
				ELSE
					//stay in this state and re-execute read
				END_IF

			ELSE
				ReadMultipleRegisters.enable := 0;
				MBError := ReadMultipleRegisters.status;
				state := MB_ERROR;
			END_IF

		MB_REQUEST_ADH_USE:

			WriteMultipleRegisters.enable := 1;
			NordsonTxPacket.Byte0_MelterControl := MelterCmd;
			NordsonTxPacket.Byte1_Command := READ_COMMAND;
			NordsonTxPacket.Byte2_Data_Index := IDX_ADHESIVE_HOUR;
			NordsonTxPacket.Byte3_Channel_Num := CHANNEL_ADHESIVE_HOUR;

			IF((WriteMultipleRegisters.status = ERR_FUB_ENABLE_FALSE) OR (WriteMultipleRegisters.status = ERR_FUB_BUSY)) THEN
				//do nothing
			ELSIF(WriteMultipleRegisters.status = ERR_OK) THEN
				WriteMultipleRegisters.enable := 0;
				state := MB_READ_ACT_TEMPS;
			ELSE
				WriteMultipleRegisters.enable := 0;
				MBError := WriteMultipleRegisters.status;
				state := MB_ERROR;
			END_IF

		MB_READ_ADH_USE:

			ReadMultipleRegisters.enable := 1;

			IF((ReadMultipleRegisters.status = ERR_FUB_ENABLE_FALSE) OR (ReadMultipleRegisters.status = ERR_FUB_BUSY)) THEN
				//do nothing
			ELSIF(ReadMultipleRegisters.status = ERR_OK) THEN
				ReadMultipleRegisters.enable := 0;

				IF((NordsonRxPacket.Byte2_Ack_Data_Index = NordsonTxPacket.Byte2_Data_Index) AND
					(NordsonRxPacket.Byte3_Ack_Channel_Num = NordsonTxPacket.Byte3_Channel_Num)) THEN

					//	NordsonData.AdhesiveUsePerHour := NordsonRxPacket.Byte4_5_Read_Data_0 + (NordsonRxPacket.Byte6_7_Read_Data_1*(65536)); //data 0 + data 1 shifted up 16 bits

					state := MB_READ_ACT_TEMPS;
				ELSE
					//stay in this state and re-execute read
				END_IF
			END_IF

		MB_WRITE_REGISTERS:

			WriteMultipleRegisters.enable := 1;
			NordsonTxPacket.Byte0_MelterControl := MELTER_ON;
			NordsonTxPacket.Byte1_Command := READ_COMMAND;
			NordsonTxPacket.Byte2_Data_Index := testChannel;
			NordsonTxPacket.Byte3_Channel_Num := testIdx;

			IF((WriteMultipleRegisters.status = ERR_FUB_ENABLE_FALSE) OR (WriteMultipleRegisters.status = ERR_FUB_BUSY)) THEN
				//do nothing
			ELSIF(WriteMultipleRegisters.status = ERR_OK) THEN
				WriteMultipleRegisters.enable := 0;
				state := MB_READ_ACT_TEMPS;
			ELSE
				WriteMultipleRegisters.enable := 0;
				MBError := WriteMultipleRegisters.status;
				state := MB_ERROR;
			END_IF

		MB_READ_REGISTERS:

			ReadMultipleRegisters.enable := 1;

			IF((ReadMultipleRegisters.status = ERR_FUB_ENABLE_FALSE) OR (ReadMultipleRegisters.status = ERR_FUB_BUSY)) THEN
				//do nothing
			ELSIF(ReadMultipleRegisters.status = ERR_OK) THEN
				ReadMultipleRegisters.enable := 0;
				state := MB_IDLE;
			ELSE
				ReadMultipleRegisters.enable := 0;
				MBError := ReadMultipleRegisters.status;
				state := MB_ERROR;
			END_IF

		MB_ERROR:
			gAdhesiveCtrlInterface.Parameters.NordsonComms.ConsecutiveErrorCount := gAdhesiveCtrlInterface.Parameters.NordsonComms.ConsecutiveErrorCount + 1;
		state := MB_IDLE; //keep re-trying indefinetly, logic below will set/reset alarms alarm

	END_CASE;

	IF EDGEPOS(gAdhesiveCtrlInterface.Parameters.NordsonComms.ConsecutiveErrorCount >= 10) THEN
		MpAlarmXSet(gAlarmXCore, ALARM_NORDSON_COMMS);
	ELSIF EDGENEG(gAdhesiveCtrlInterface.Parameters.NordsonComms.ConsecutiveErrorCount >= 10)THEN
		MpAlarmXReset(gAlarmXCore, ALARM_NORDSON_COMMS);
	END_IF

	IF EDGEPOS(gAdhesiveCtrlInterface.Status.ATS_AddOnOverLimit) THEN
		MpAlarmXSet(gAlarmXCore, ALARM_ATS_OVERLIMIT);
	ELSIF EDGENEG(gAdhesiveCtrlInterface.Status.ATS_AddOnOverLimit)THEN
		MpAlarmXReset(gAlarmXCore, ALARM_ATS_OVERLIMIT);
	END_IF

	IF EDGEPOS(gAdhesiveCtrlInterface.Status.ATS_AddOnUnderLimit) THEN
		MpAlarmXSet(gAlarmXCore, ALARM_ATS_UNDERLIMIT);
	ELSIF EDGENEG(gAdhesiveCtrlInterface.Status.ATS_AddOnUnderLimit)THEN
		MpAlarmXReset(gAlarmXCore, ALARM_ATS_UNDERLIMIT);
	END_IF

	IF EDGEPOS(gAdhesiveCtrlInterface.Status.NordsonInStandby) THEN
		MpAlarmXSet(gAlarmXCore, ALARM_NORDSON_STANDBY);
	ELSIF EDGENEG(gAdhesiveCtrlInterface.Status.NordsonInStandby)THEN
		MpAlarmXReset(gAlarmXCore, ALARM_NORDSON_STANDBY);
	END_IF

	//force unit ready and unit faulted status flags if ModbusTCP control is selected and bypass is enabled
	IF(gAdhesiveCtrlInterface.Parameters.FeedbackIsModbusTCP AND gAdhesiveCtrlInterface.Parameters.NordsonComms.ByPassFeedback) THEN
		gAdhesiveCtrlInterface.Parameters.NordsonComms.UnitReady := TRUE;
		gAdhesiveCtrlInterface.Parameters.NordsonComms.UnitFaulted := FALSE;
		gAdhesiveCtrlInterface.Status.ATS_AddOnOverLimit := FALSE;
		gAdhesiveCtrlInterface.Status.ATS_AddOnUnderLimit := FALSE;
	END_IF

	//Must be called after state machine. Do not move any function calls that are already below this line
	WriteMultipleRegisters.pStation := ADR(mb_station);
	WriteMultipleRegisters.startAddress := write_register_address;
	WriteMultipleRegisters.nrRegisters := num_registers_to_write;
	WriteMultipleRegisters.pData := ADR(NordsonTxPacket);
	WriteMultipleRegisters.dataSize := SIZEOF(NordsonTxPacket);
	WriteMultipleRegisters();

	ReadMultipleRegisters.pStation := ADR(mb_station);
	ReadMultipleRegisters.startAddress := read_register_address;
	ReadMultipleRegisters.nrRegisters := num_registers_to_read;
	ReadMultipleRegisters.pData := ADR(NordsonRxPacket);
	ReadMultipleRegisters.dataSize := SIZEOF(NordsonRxPacket);
	ReadMultipleRegisters();

	FeedbackCycleTimer.PT := gAdhesiveCtrlInterface.Parameters.NordsonComms.FeedbackTime;
	FeedbackCycleTimer();

				END_PROGRAM
```

### Data object Logical/gFeedobj/gFeedi (Ax)

#### gFeedi.ax
```
InitParameter (Version=5.08.2, NcSwId=ACP10)
  ACP10AXIS_typ:
    dig_in:
      level:
        reference = ncACTIV_HI
        pos_hw_end = ncACTIV_HI
        neg_hw_end = ncACTIV_HI
        trigger1 = ncACTIV_HI
        trigger2 = ncACTIV_HI
    encoder_if:
      parameter:
        count_dir = ncSTANDARD
        scaling:
          load:
            units = 2651125
            rev_motor = 793
    limit:
      parameter:
        v_pos = 139100.0
        v_neg = 139100.0
        a1_pos = 305500.0
        a2_pos = 305500.0
        a1_neg = 305500.0
        a2_neg = 305500.0
        t_jolt = 0.0
        t_in_pos = 0.0
        pos_sw_end = 110000
        neg_sw_end = 0
        ds_warning = 1200.0
        ds_stop = 1200.0
        a_stop = 1.0E+30
        dv_stop = 0.0
        dv_stop_mode = ncOFF
    controller:
      mode = ncPOSITION
      position:
        kv = 250.0
        tn = 0.0
        t_predict = 0.0004
        t_total = 0.0004
        p_max = 1.0E+30
        i_max = 1.0E+30
      speed:
        kv = 7.5
        tn = 0.1
        t_filter = 0.0
        isq_filter1:
          type = ncOFF
          a0 = 0.0
          a1 = 0.0
          b0 = 0.0
          b1 = 0.0
          b2 = 0.0
          c0_par_id = 0
          c1_par_id = 0
        isq_filter2:
          type = ncOFF
          a0 = 0.0
          a1 = 0.0
          b0 = 0.0
          b1 = 0.0
          b2 = 0.0
          c0_par_id = 0
          c1_par_id = 0
        isq_filter3:
          type = ncOFF
          a0 = 0.0
          a1 = 0.0
          b0 = 0.0
          b1 = 0.0
          b2 = 0.0
          c0_par_id = 0
          c1_par_id = 0
      uf:
        type = ncLINEAR
        auto_config = ncOFF
        u0 = 0.0
        un = 0.0
        fn = 0.0
        k_f_slip = 0.0
      ff:
        mode = ncSTANDARD
        torque_load = 0.0
        torque_pos = 0.0
        torque_neg = 0.0
        kv_torque = 0.0
        inertia = 0.0
        t_filter_a = 0.0
      fb:
        mode = ncSTANDARD
        speed_mix_ratio = 0.0
        speed_kv = 2.0
      model:
        mass1:
          inertia = 0.0
          viscous_friction = 0.0
        mass2:
          inertia = 0.0
          viscous_friction = 0.0
          stiffness = 0.0
          damping = 0.0
    move:
      stop:
        parameter[0]:
          decel_ramp = ncA_LIMIT
          controller = ncON
        parameter[1]:
          decel_ramp = ncA_LIMIT
          controller = ncON
        parameter[2]:
          decel_ramp = ncA_LIMIT
          controller = ncON
        parameter[3]:
          decel_ramp = ncA_LIMIT
          controller = ncON
        quickstop:
          decel_ramp = ncA_LIMIT
          t_jolt = 0.0
        drive_error:
          decel_ramp = ncA_LIMIT
      homing:
        parameter:
          s = -1250
          v_switch = 1000.0
          v_trigger = 500.0
          a = 50000.0
          mode = ncBLOCK_DS
          edge_sw = ncPOSITIVE
          start_dir = ncNEGATIVE
          trigg_dir = ncPOSITIVE
          ref_pulse = ncOFF
          fix_dir = ncOFF
          tr_s_block = 0.0
          torque_lim = 8.0
          ds_block = 150.0
          ds_stop = 200.0
      basis:
        parameter:
          v_pos = 10000.0
          v_neg = 10000.0
          a1_pos = 140000.0
          a2_pos = 140000.0
          a1_neg = 140000.0
          a2_neg = 140000.0
    message:
      text:
        parameter:
          format = ncBREAK
          columns = 80
          data_modul = acp10etxen
```

### Data object Logical/gFeedobj/brake (Apt)

#### AcpParTab.apt
```
AcoposParameterTable:
  Root Parameters:
    8B0W0026H000.A00-1 mounting horizontal V1:
      Group (Disabled=TRUE)  //  DO NOT USE with ACOPOS Firmware before V2.27.0
      10 = 360 (Name=R_BLEEDER_EXT, Unit=Ohm, Disabled=FALSE)  // Bleeder: External: Resistance
      11 = 380 (Name=TEMP_MAX_BLEEDER_EXT, Unit=°C, Disabled=FALSE)  // Bleeder: External: Limit temperature
      12 = 2.54 (Name=RTH_BLEEDER_AMB_EXT, Unit=K/W, Disabled=FALSE)  // Bleeder: External: Thermic resistance
      13 = 2.38 (Name=CTH_BLEEDER_EXT, Unit=Ws/K, Disabled=FALSE)  // Bleeder: External: Thermic capacity
      398 = 1 (Name=BLEEDER_SELECTOR_EXT, Disabled=FALSE)  // Bleeder: Selector
      866 = 64 (Name=MOTOR_TEST_MODE)  // Motor: Test mode
```

- Data object Logical/gFeedobj/disablebrakecheck (Apt) (no source held here)

### Program Logical/HMI/HMIControl

#### Cyclic.ld
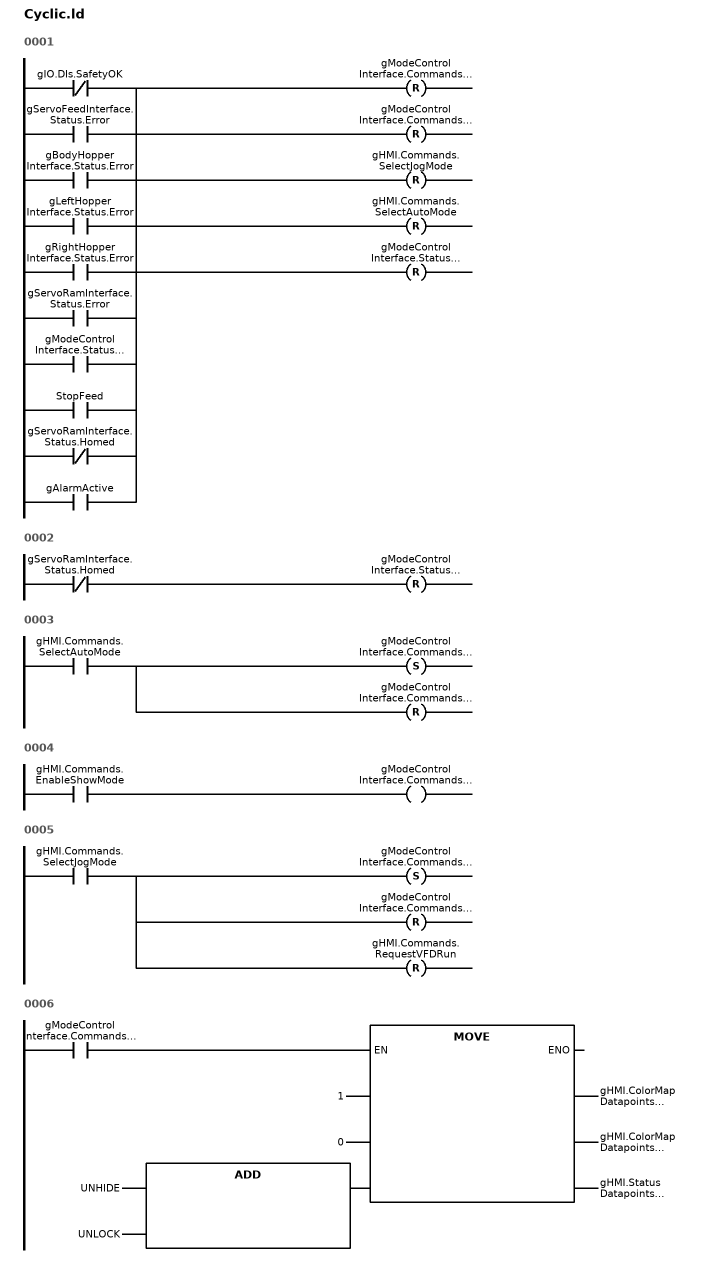
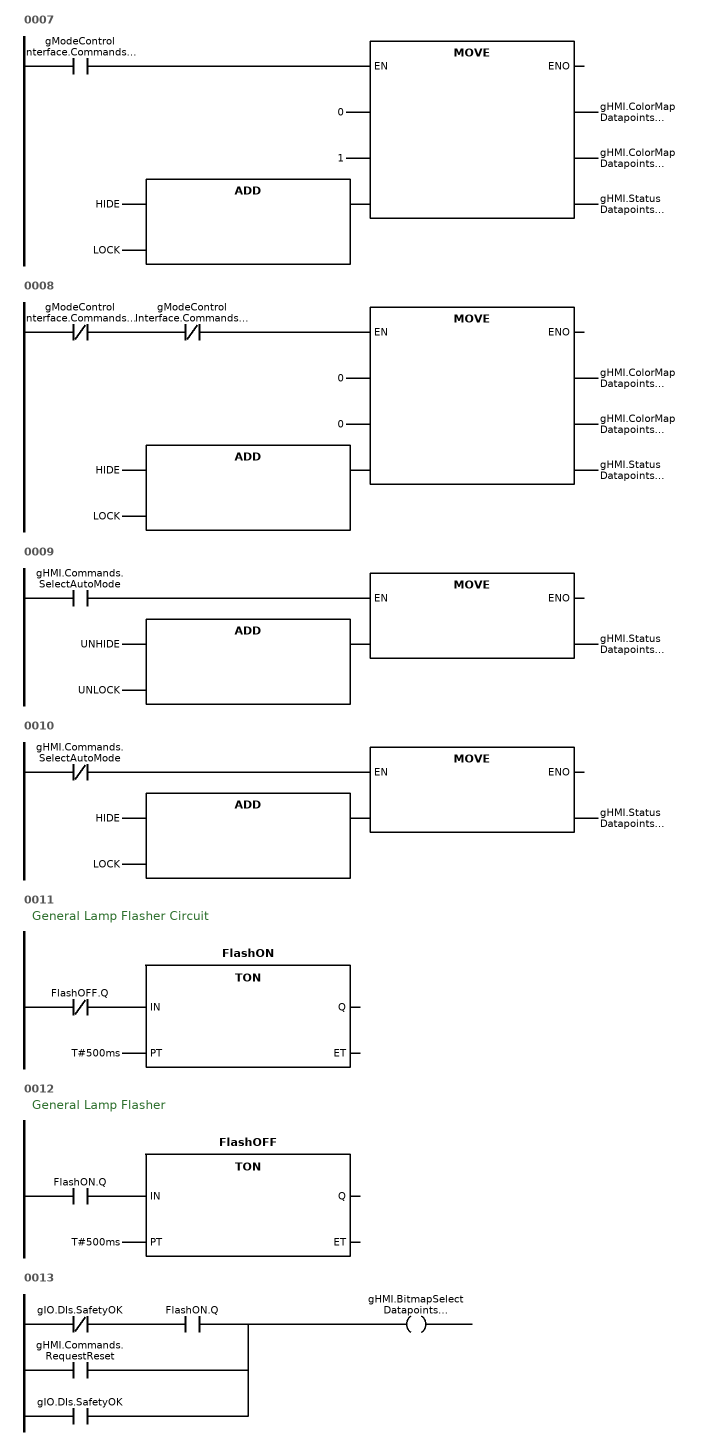
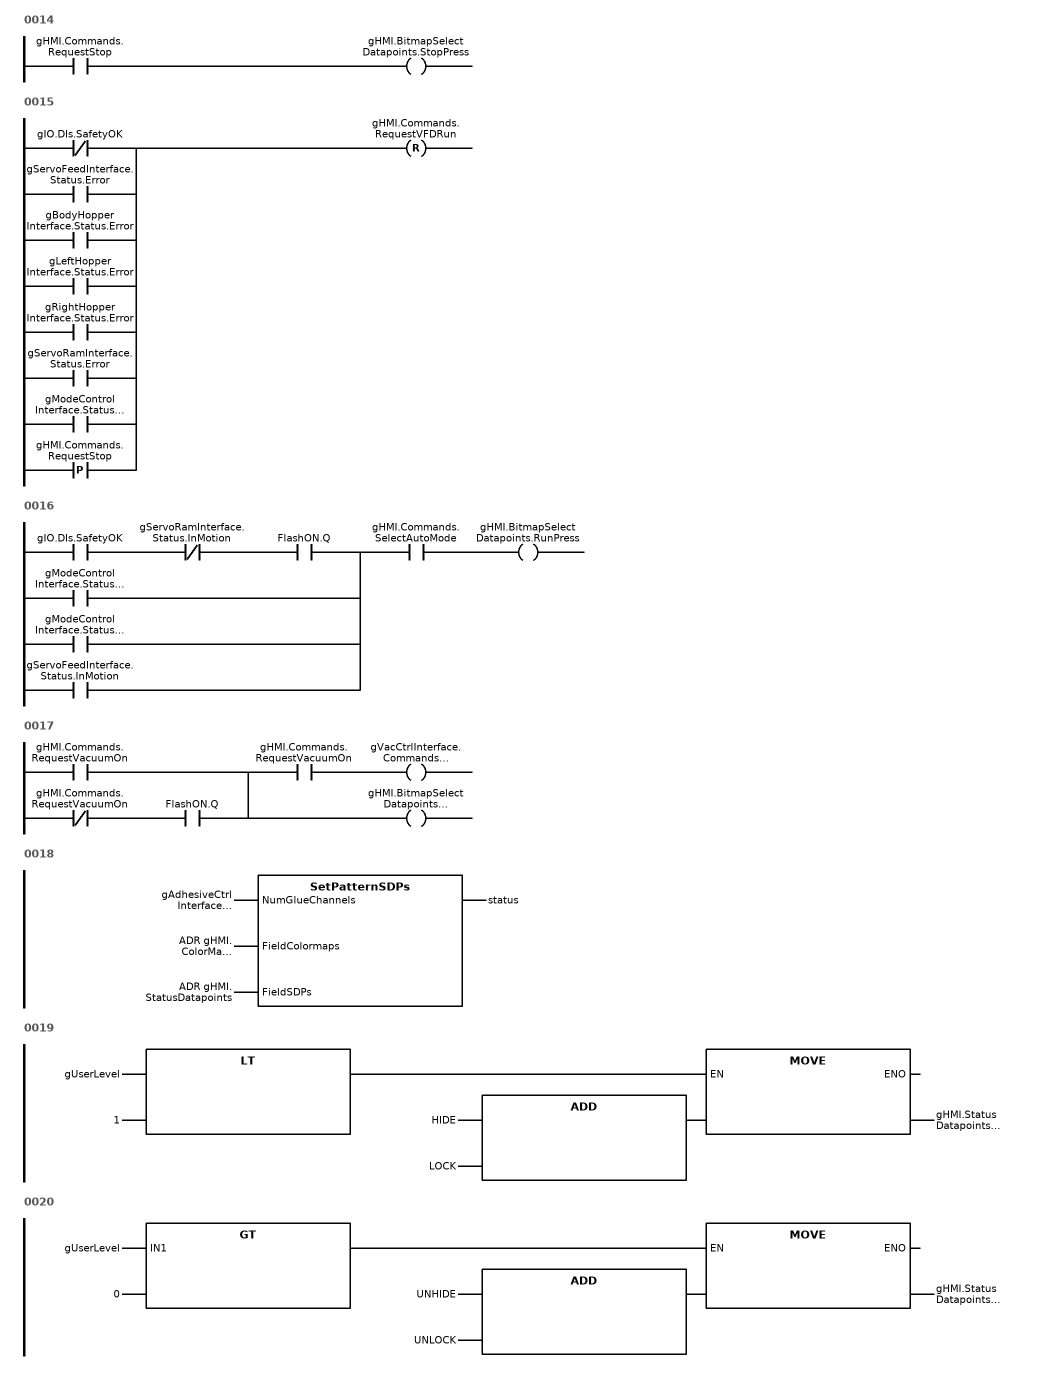
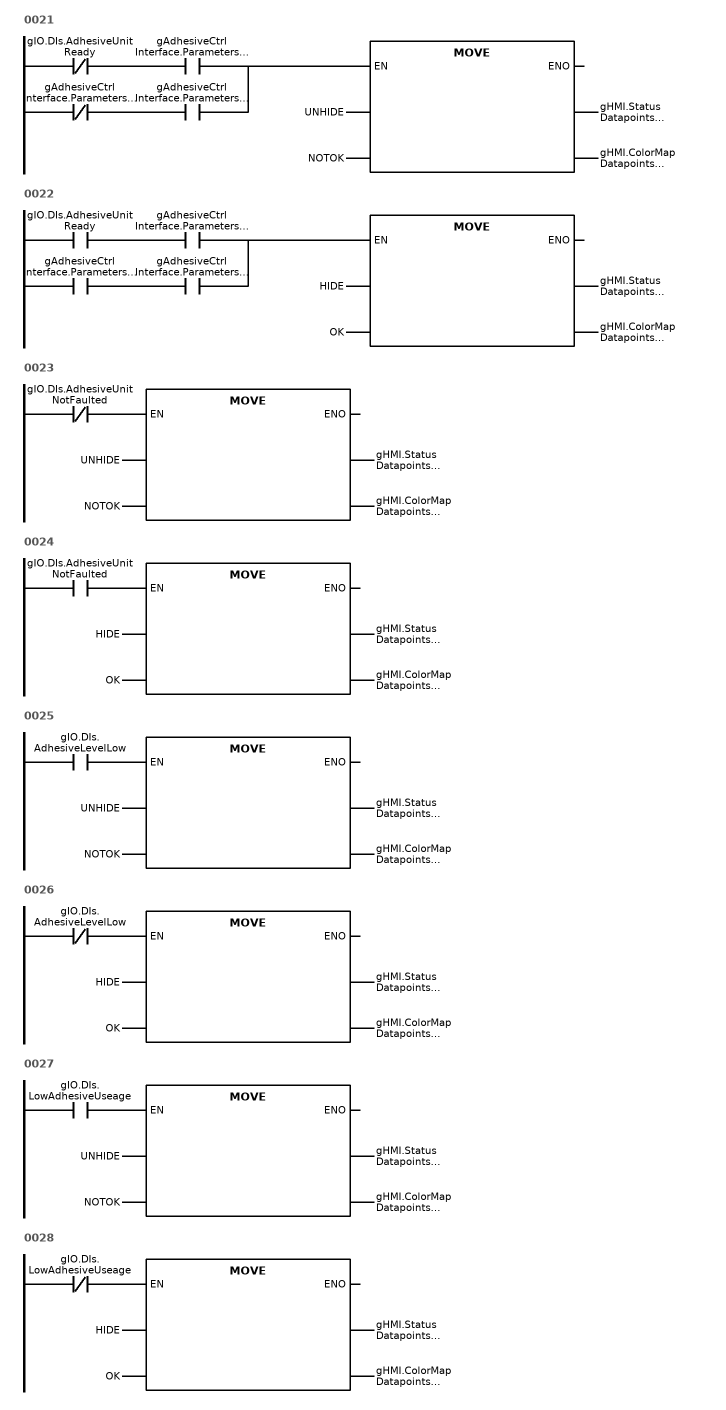
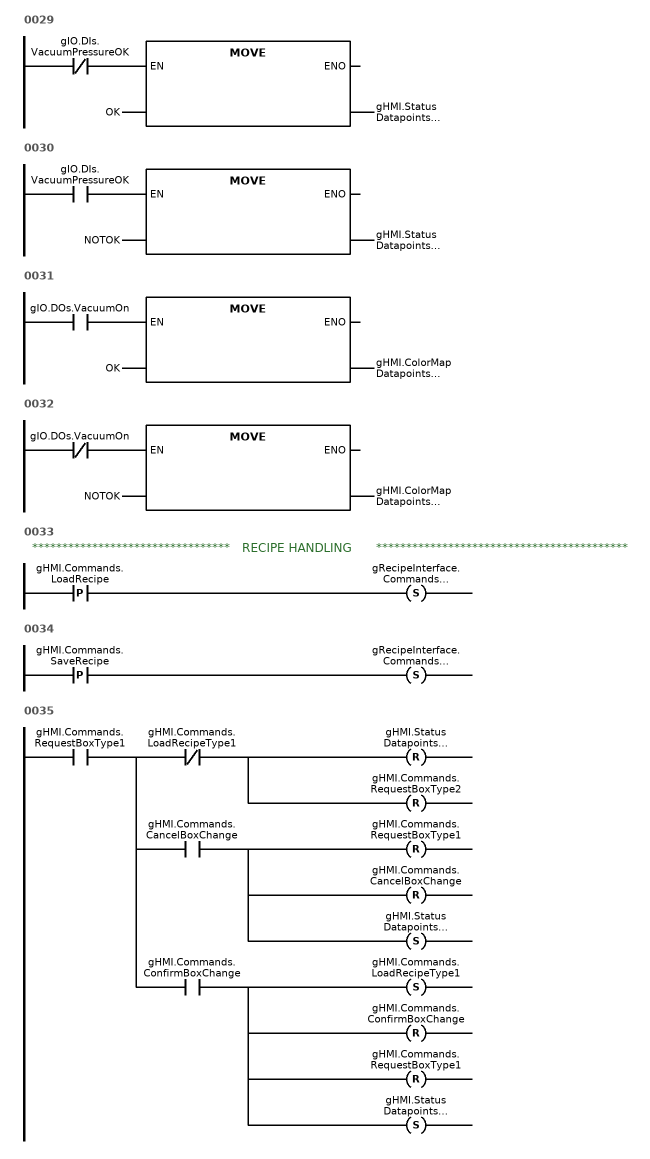
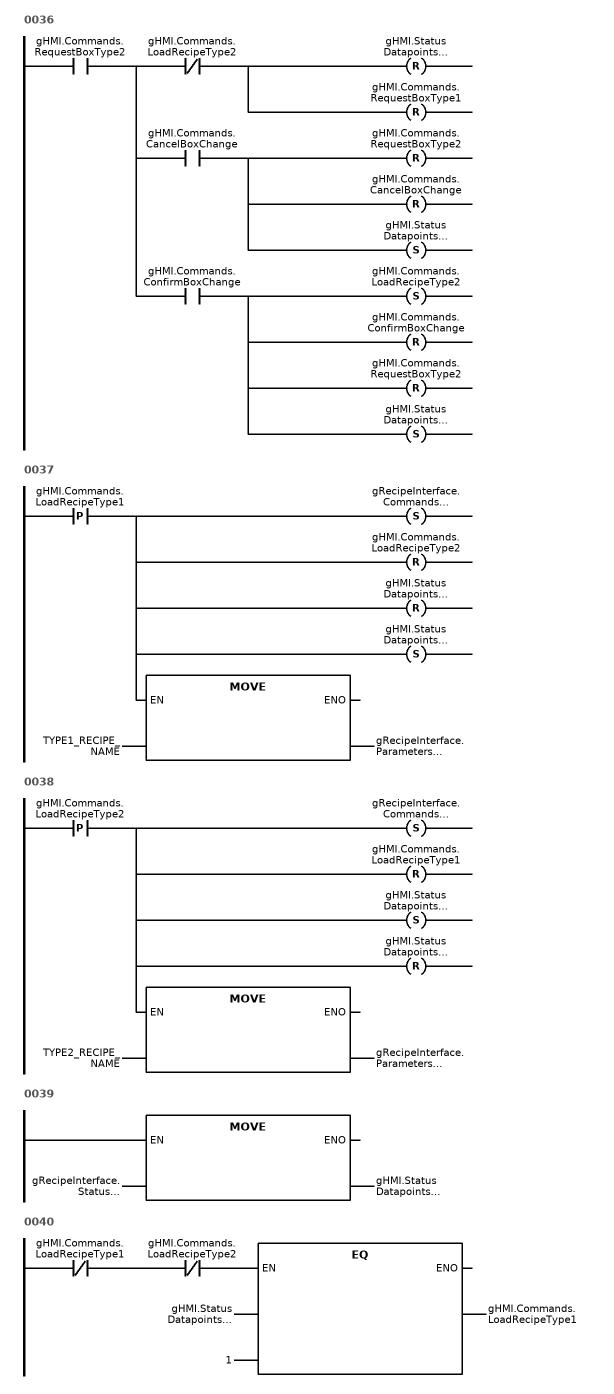
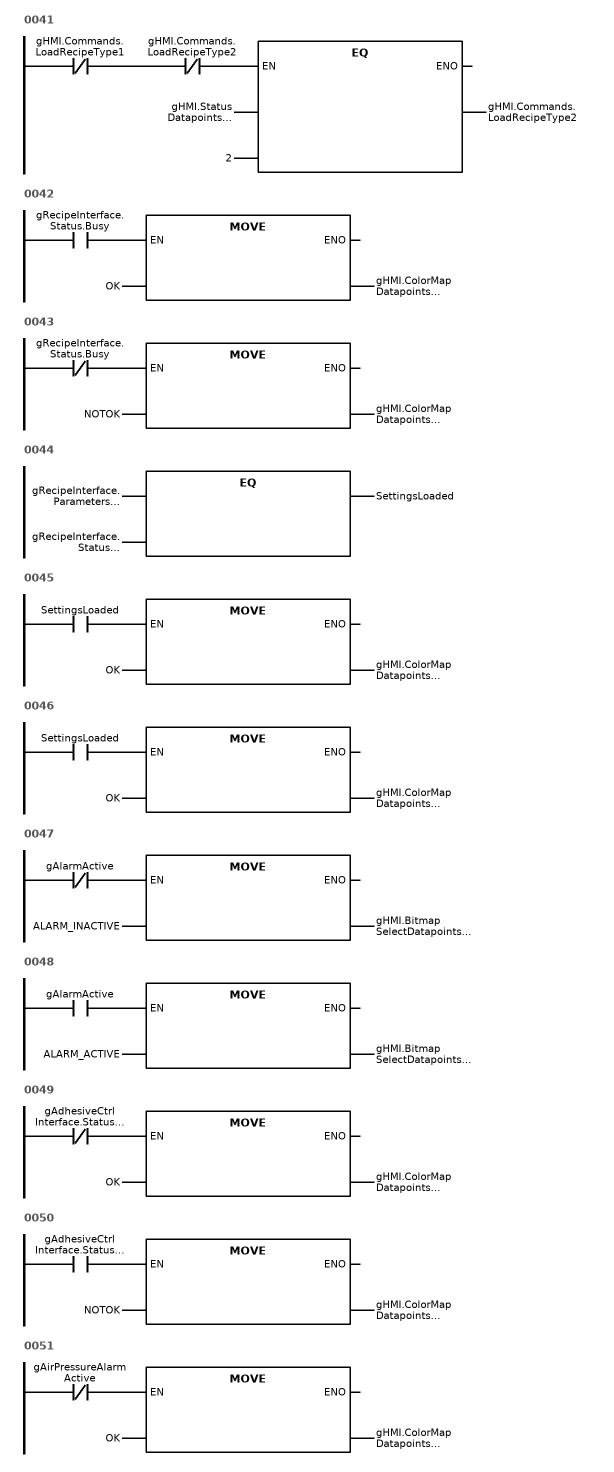
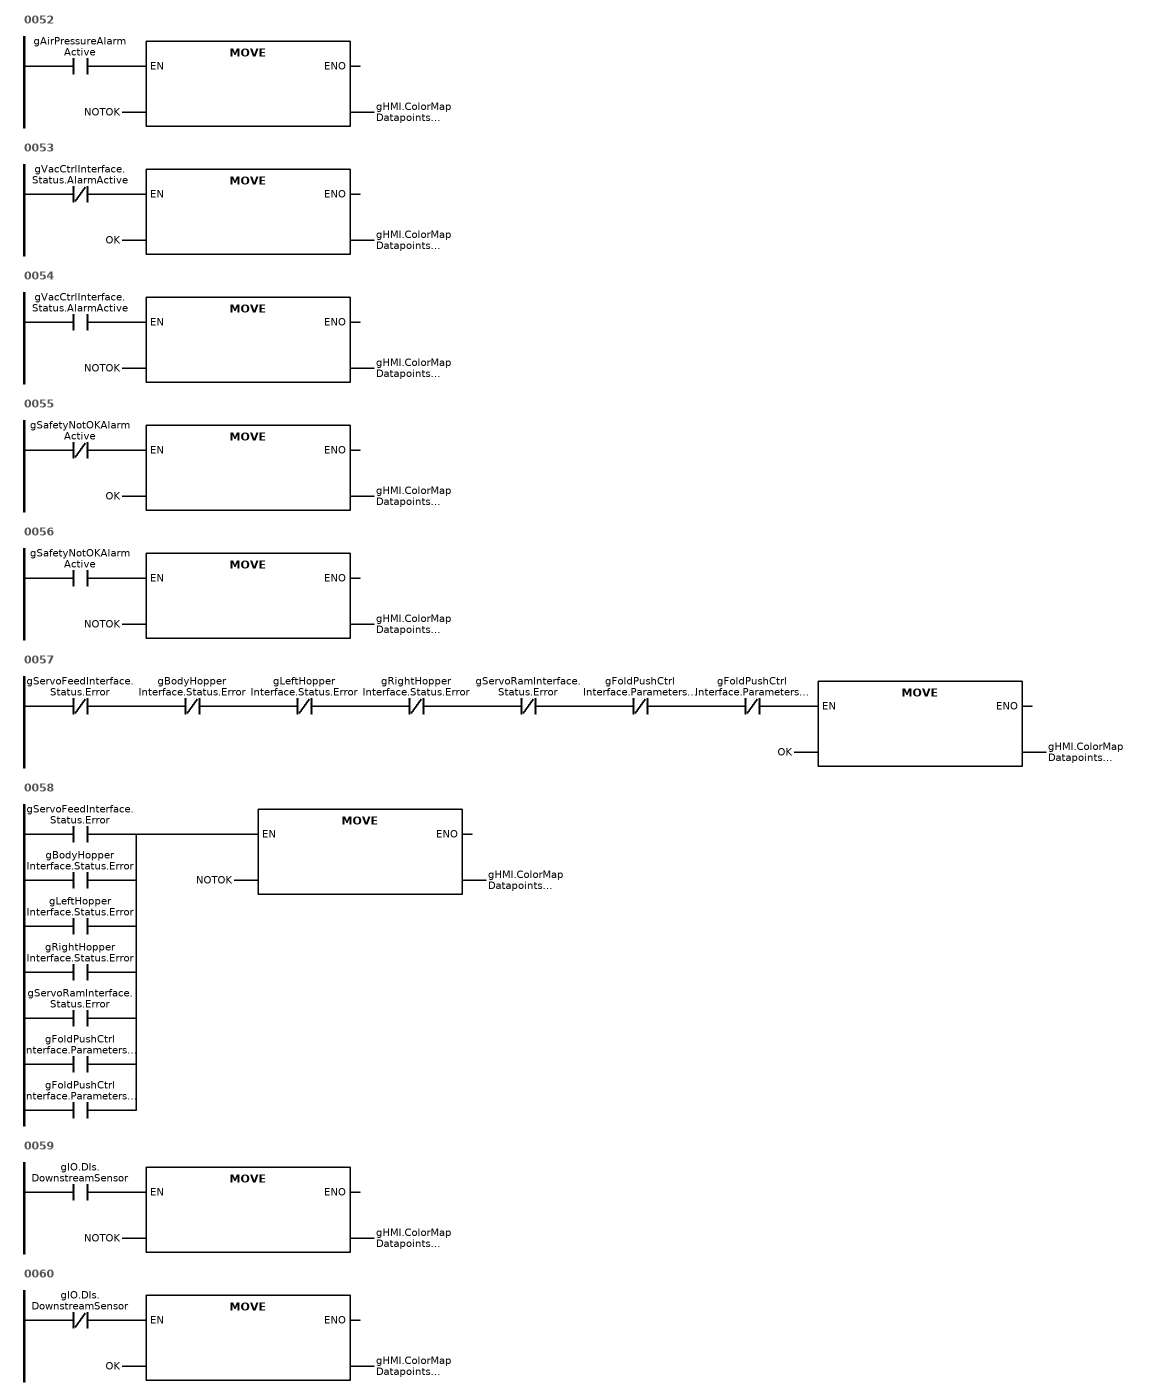
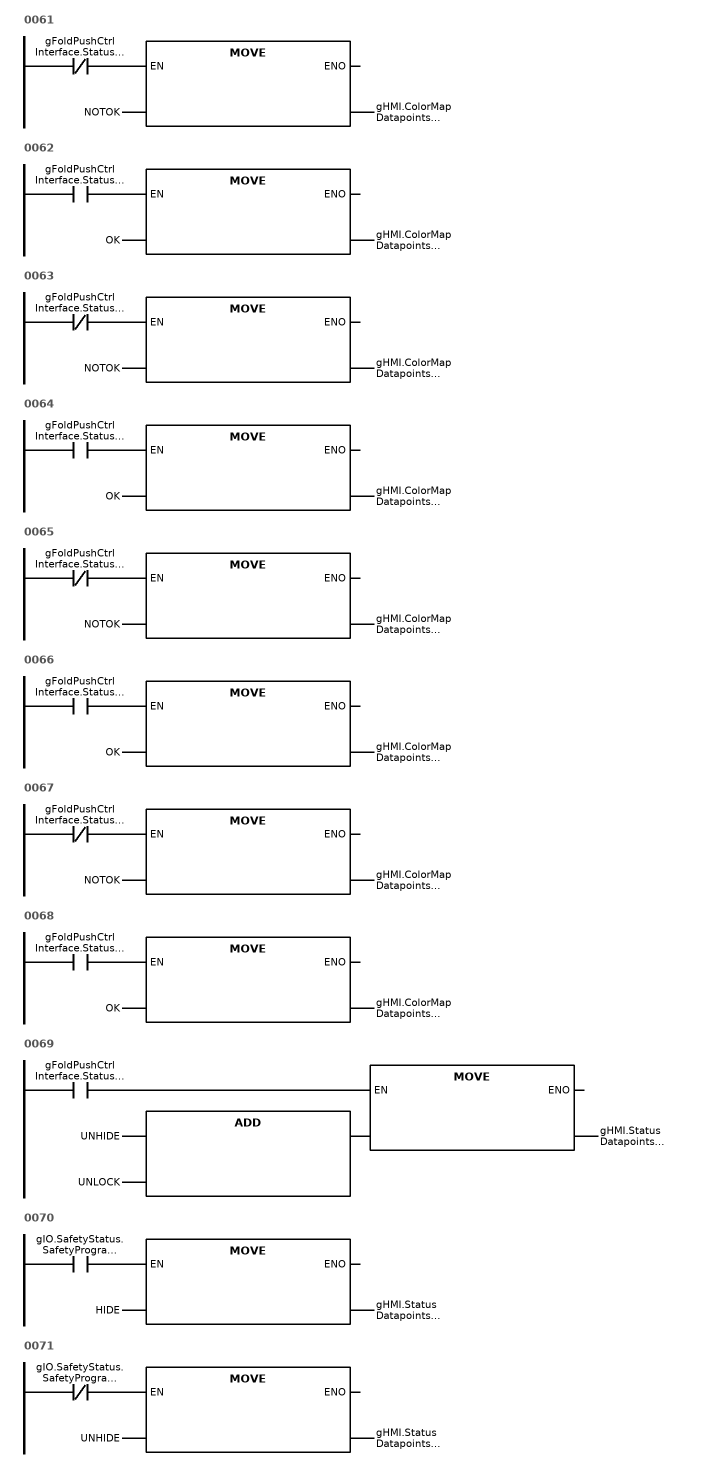
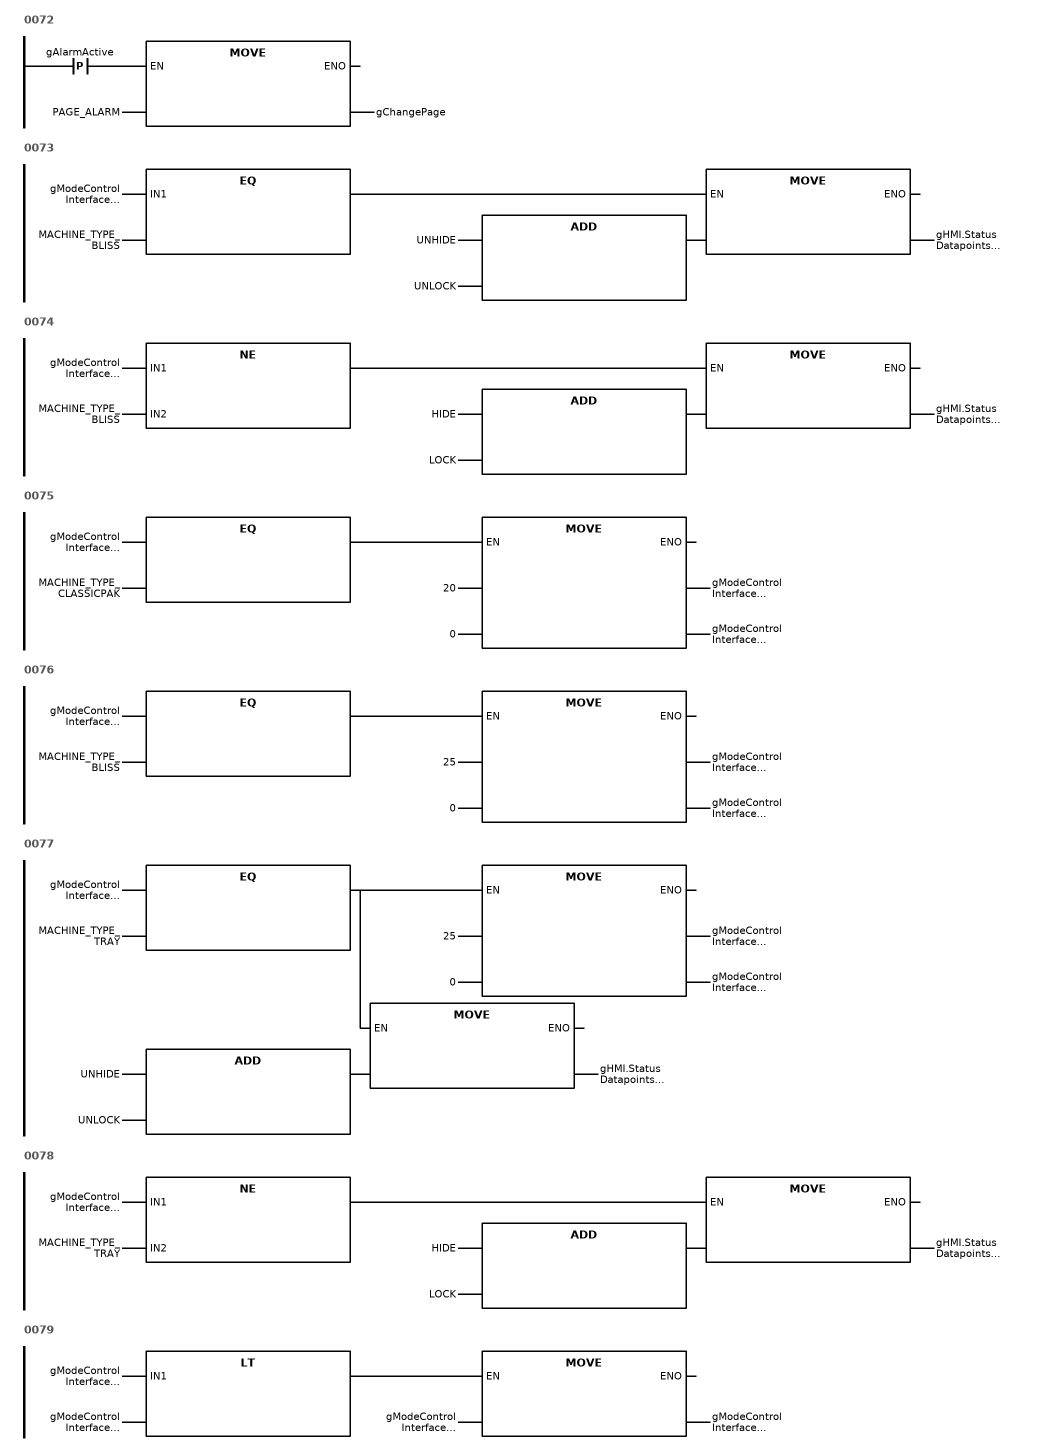
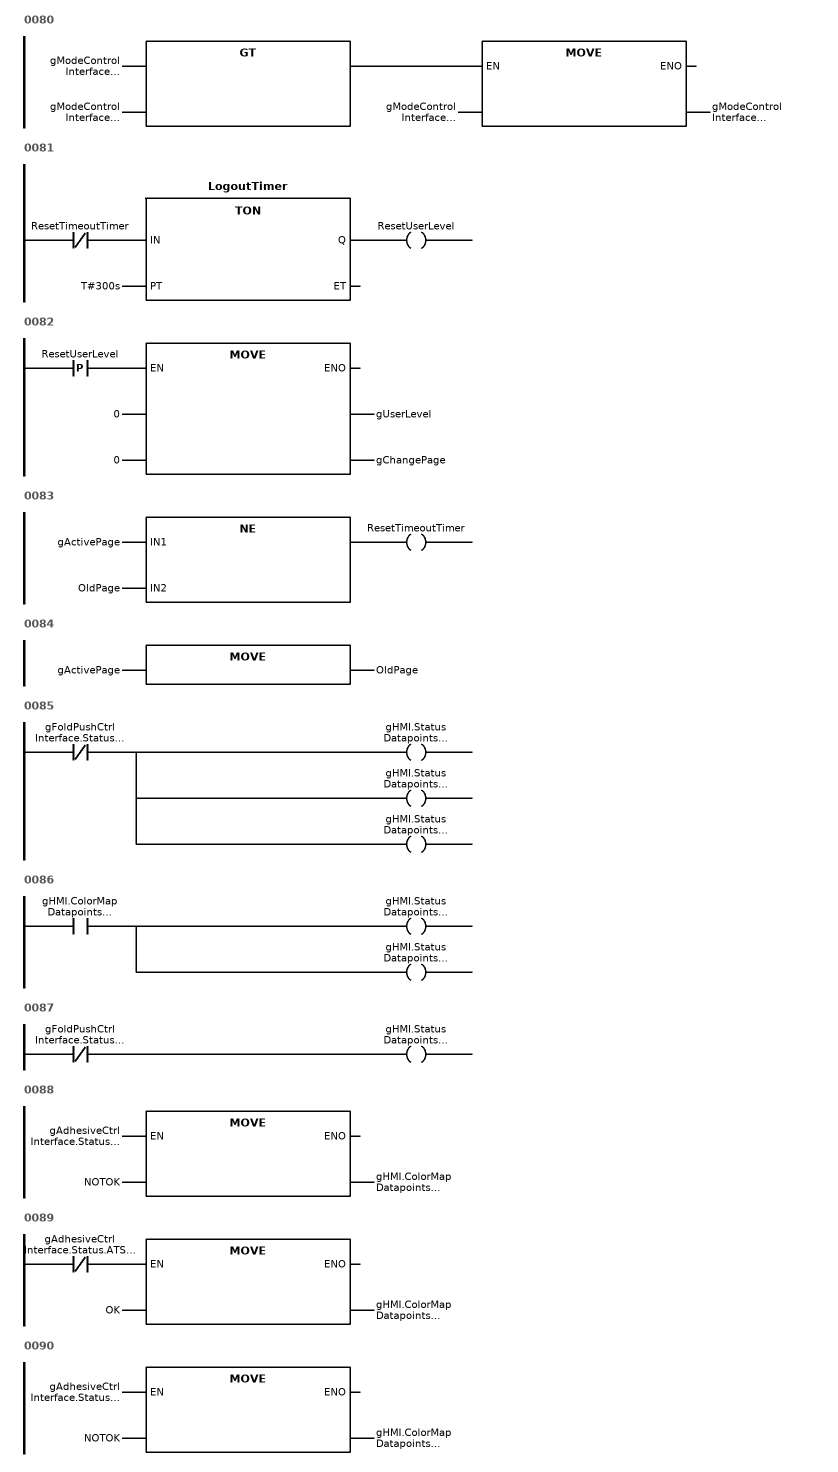
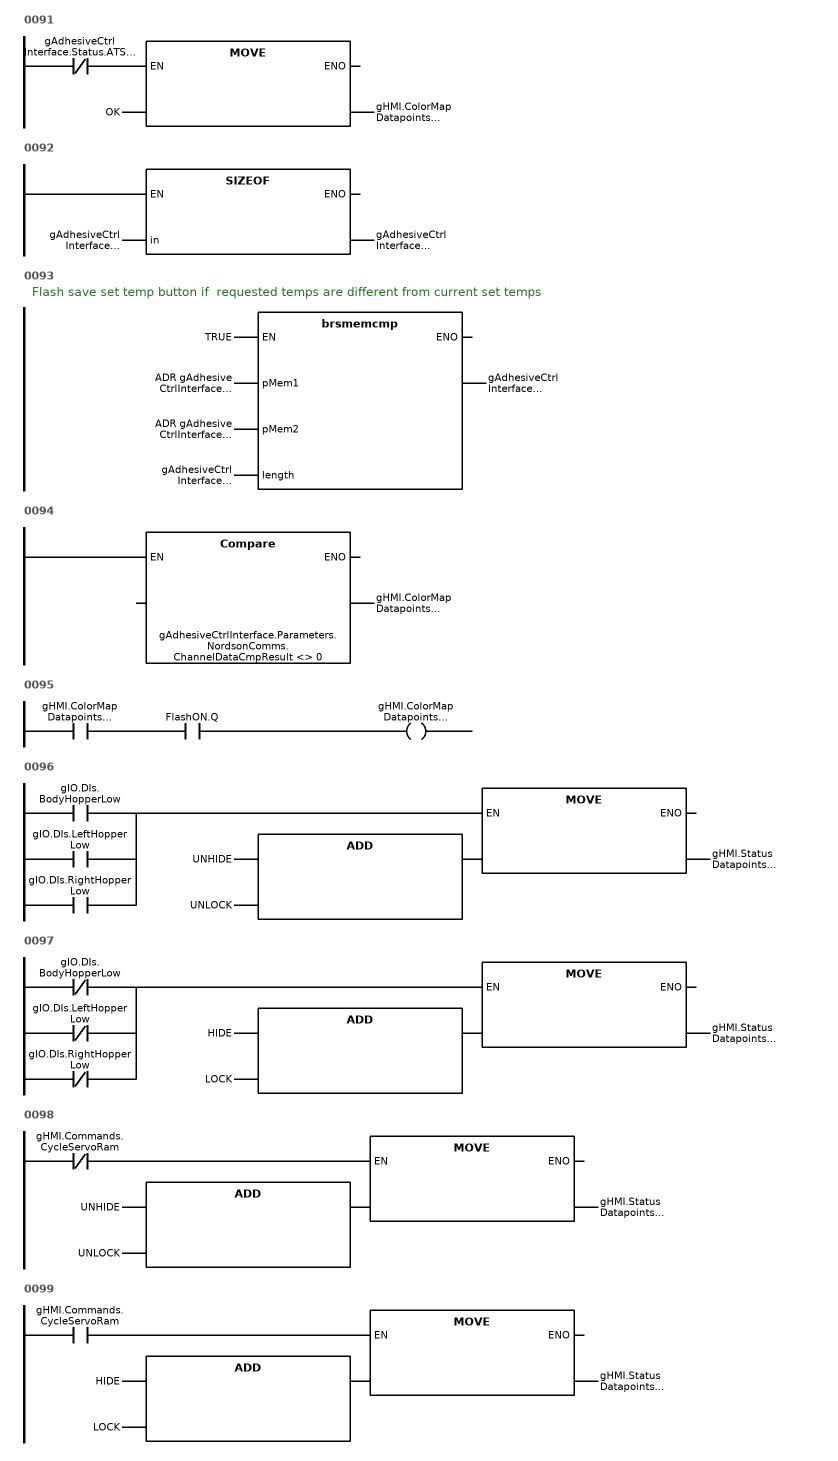
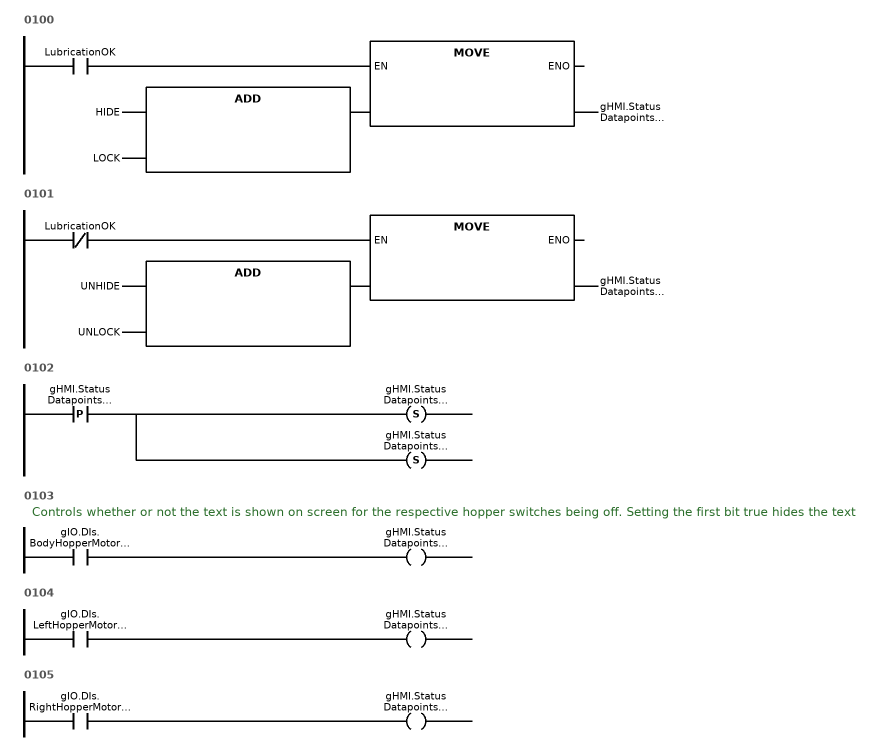
Ladder, written as Structured Text:
```iecst
PROGRAM _CYCLIC
VAR
    _p1 : BOOL;
    _p2 : BOOL;
    _p3 : BOOL;
    _p4 : BOOL;
    _e5 : R_TRIG;
    _p6 : BOOL;
    _p7 : BOOL;
    _p8 : BOOL;
    _p9 : BOOL;
    _e10 : R_TRIG;
    _e11 : R_TRIG;
    _p12 : BOOL;
    _p13 : BOOL;
    _p14 : BOOL;
    _p15 : BOOL;
    _p16 : BOOL;
    _p17 : BOOL;
    _p18 : BOOL;
    _p19 : BOOL;
    _e20 : R_TRIG;
    _e21 : R_TRIG;
    _p22 : BOOL;
    _p23 : BOOL;
    _e24 : R_TRIG;
    _t25 : BOOL;
    _t26 : BOOL;
    _t27 : BOOL;
    _p28 : BOOL;
    _p29 : BOOL;
    _e30 : R_TRIG;
    _p31 : BOOL;
    _p32 : BOOL;
    _p33 : BOOL;
    _e34 : R_TRIG;
END_VAR
(* Network 1 *)
_p1 := gModeControlInterface.Status.BlissPanelAlarmActive;
IF NOT gIO.DIs.SafetyOK OR gServoFeedInterface.Status.Error OR gBodyHopperInterface.Status.Error OR gLeftHopperInterface.Status.Error OR gRightHopperInterface.Status.Error OR gServoRamInterface.Status.Error OR _p1 OR StopFeed OR NOT gServoRamInterface.Status.Homed OR gAlarmActive THEN
    gModeControlInterface.Commands.SetAutoMode := FALSE;
    gModeControlInterface.Commands.SetJogMode := FALSE;
    gHMI.Commands.SelectJogMode := FALSE;
    gHMI.Commands.SelectAutoMode := FALSE;
    gModeControlInterface.Status.Dwelling := FALSE;
END_IF;

(* Network 2 *)
IF NOT gServoRamInterface.Status.Homed THEN gModeControlInterface.Status.Dwelling := FALSE; END_IF;

(* Network 3 *)
IF gHMI.Commands.SelectAutoMode THEN
    gModeControlInterface.Commands.SetAutoMode := TRUE;
    gModeControlInterface.Commands.SetJogMode := FALSE;
END_IF;

(* Network 4 *)
gModeControlInterface.Commands.SetShowMode := gHMI.Commands.EnableShowMode;

(* Network 5 *)
IF gHMI.Commands.SelectJogMode THEN
    gModeControlInterface.Commands.SetJogMode := TRUE;
    gModeControlInterface.Commands.SetAutoMode := FALSE;
    gHMI.Commands.RequestVFDRun := FALSE;
END_IF;

(* Network 6 *)
IF gModeControlInterface.Commands.SetJogMode THEN
    gHMI.ColorMapDatapoints.JogModeSelected := 1;
    gHMI.ColorMapDatapoints.AutoModeSelected := 0;
    gHMI.StatusDatapoints.JogStatusDatapoint := UNHIDE + UNLOCK;
END_IF;

(* Network 7 *)
IF gModeControlInterface.Commands.SetAutoMode THEN
    gHMI.ColorMapDatapoints.JogModeSelected := 0;
    gHMI.ColorMapDatapoints.AutoModeSelected := 1;
    gHMI.StatusDatapoints.JogStatusDatapoint := HIDE + LOCK;
END_IF;

(* Network 8 *)
_p2 := NOT gModeControlInterface.Commands.SetAutoMode AND NOT gModeControlInterface.Commands.SetJogMode;
IF _p2 THEN
    gHMI.ColorMapDatapoints.JogModeSelected := 0;
    gHMI.ColorMapDatapoints.AutoModeSelected := 0;
    gHMI.StatusDatapoints.JogStatusDatapoint := HIDE + LOCK;
END_IF;

(* Network 9 *)
_p3 := gHMI.Commands.SelectAutoMode;
IF _p3 THEN gHMI.StatusDatapoints.AutoModeSDP := UNHIDE + UNLOCK; END_IF;

(* Network 10 *)
_p4 := NOT gHMI.Commands.SelectAutoMode;
IF _p4 THEN gHMI.StatusDatapoints.AutoModeSDP := HIDE + LOCK; END_IF;

(* Network 11: General Lamp Flasher Circuit *)
FlashON(IN := NOT FlashOFF.Q, PT := T#500ms);

(* Network 12: General Lamp Flasher *)
FlashOFF(IN := FlashON.Q, PT := T#500ms);

(* Network 13 *)
gHMI.BitmapSelectDatapoints.ResetPress := (NOT gIO.DIs.SafetyOK AND FlashON.Q) OR gHMI.Commands.RequestReset OR gIO.DIs.SafetyOK;

(* Network 14 *)
gHMI.BitmapSelectDatapoints.StopPress := gHMI.Commands.RequestStop;

(* Network 15 *)
_e5(CLK := gHMI.Commands.RequestStop);
IF NOT gIO.DIs.SafetyOK OR gServoFeedInterface.Status.Error OR gBodyHopperInterface.Status.Error OR gLeftHopperInterface.Status.Error OR gRightHopperInterface.Status.Error OR gServoRamInterface.Status.Error OR gModeControlInterface.Status.BlissPanelAlarmActive OR _e5.Q THEN
    gHMI.Commands.RequestVFDRun := FALSE;
END_IF;

(* Network 16 *)
gHMI.BitmapSelectDatapoints.RunPress := ((gIO.DIs.SafetyOK AND NOT gServoRamInterface.Status.InMotion AND FlashON.Q) OR gModeControlInterface.Status.Dwelling OR gModeControlInterface.Status.WaitingOnDownstream OR gServoFeedInterface.Status.InMotion) AND gHMI.Commands.SelectAutoMode;

(* Network 17 *)
gVacCtrlInterface.Commands.VacuumOn := (gHMI.Commands.RequestVacuumOn OR (NOT gHMI.Commands.RequestVacuumOn AND FlashON.Q)) AND gHMI.Commands.RequestVacuumOn;
gHMI.BitmapSelectDatapoints.VacuumPress := gHMI.Commands.RequestVacuumOn OR (NOT gHMI.Commands.RequestVacuumOn AND FlashON.Q);

(* Network 18 *)
status := SetPatternSDPs(NumGlueChannels := gAdhesiveCtrlInterface.Parameters.NumAdhesiveChannels, FieldColormaps := ADR(gHMI.ColorMapDatapoints), FieldSDPs := ADR(gHMI.StatusDatapoints));

(* Network 19 *)
IF gUserLevel < 1 THEN gHMI.StatusDatapoints.MaintenanceSDP := HIDE + LOCK; END_IF;

(* Network 20 *)
IF gUserLevel > 0 THEN gHMI.StatusDatapoints.MaintenanceSDP := UNHIDE + UNLOCK; END_IF;

(* Network 21 *)
_p6 := NOT gIO.DIs.AdhesiveUnitReady AND gAdhesiveCtrlInterface.Parameters.FeedbackIsHardwire;
_p7 := NOT gAdhesiveCtrlInterface.Parameters.NordsonComms.UnitReady AND gAdhesiveCtrlInterface.Parameters.FeedbackIsModbusTCP;
IF _p6 OR _p7 THEN
    gHMI.StatusDatapoints.AdhesiveUnitNotReadySDP := UNHIDE;
    gHMI.ColorMapDatapoints.AdhesiveUnitReady := NOTOK;
END_IF;

(* Network 22 *)
_p8 := gIO.DIs.AdhesiveUnitReady AND gAdhesiveCtrlInterface.Parameters.FeedbackIsHardwire;
_p9 := gAdhesiveCtrlInterface.Parameters.NordsonComms.UnitReady AND gAdhesiveCtrlInterface.Parameters.FeedbackIsModbusTCP;
IF _p8 OR _p9 THEN
    gHMI.StatusDatapoints.AdhesiveUnitNotReadySDP := HIDE;
    gHMI.ColorMapDatapoints.AdhesiveUnitReady := OK;
END_IF;

(* Network 23 *)
IF NOT gIO.DIs.AdhesiveUnitNotFaulted THEN
    gHMI.StatusDatapoints.AdhesiveUnitFaultSDP := UNHIDE;
    gHMI.ColorMapDatapoints.AdhesiveUnitFault := NOTOK;
END_IF;

(* Network 24 *)
IF gIO.DIs.AdhesiveUnitNotFaulted THEN
    gHMI.StatusDatapoints.AdhesiveUnitFaultSDP := HIDE;
    gHMI.ColorMapDatapoints.AdhesiveUnitFault := OK;
END_IF;

(* Network 25 *)
IF gIO.DIs.AdhesiveLevelLow THEN
    gHMI.StatusDatapoints.AdhesiveUnitLevelLowSDP := UNHIDE;
    gHMI.ColorMapDatapoints.AdhesiveUnitLevelLow := NOTOK;
END_IF;

(* Network 26 *)
IF NOT gIO.DIs.AdhesiveLevelLow THEN
    gHMI.StatusDatapoints.AdhesiveUnitLevelLowSDP := HIDE;
    gHMI.ColorMapDatapoints.AdhesiveUnitLevelLow := OK;
END_IF;

(* Network 27 *)
IF gIO.DIs.LowAdhesiveUseage THEN
    gHMI.StatusDatapoints.AdhesiveUseageLowSDP := UNHIDE;
    gHMI.ColorMapDatapoints.AdhesiveUseageLow := NOTOK;
END_IF;

(* Network 28 *)
IF NOT gIO.DIs.LowAdhesiveUseage THEN
    gHMI.StatusDatapoints.AdhesiveUseageLowSDP := HIDE;
    gHMI.ColorMapDatapoints.AdhesiveUseageLow := OK;
END_IF;

(* Network 29 *)
IF NOT gIO.DIs.VacuumPressureOK THEN gHMI.StatusDatapoints.VacuumPressureFaultSDP := OK; END_IF;

(* Network 30 *)
IF gIO.DIs.VacuumPressureOK THEN gHMI.StatusDatapoints.VacuumPressureFaultSDP := NOTOK; END_IF;

(* Network 31 *)
IF gIO.DOs.VacuumOn THEN gHMI.ColorMapDatapoints.VacuumPumpOn := OK; END_IF;

(* Network 32 *)
IF NOT gIO.DOs.VacuumOn THEN gHMI.ColorMapDatapoints.VacuumPumpOn := NOTOK; END_IF;

(* Network 33: *********************************   RECIPE HANDLING      ****************************************** *)
_e10(CLK := gHMI.Commands.LoadRecipe);
IF _e10.Q THEN gRecipeInterface.Commands.LoadRecipe := TRUE; END_IF;

(* Network 34 *)
_e11(CLK := gHMI.Commands.SaveRecipe);
IF _e11.Q THEN gRecipeInterface.Commands.SaveRecipe := TRUE; END_IF;

(* Network 35 *)
_p12 := gHMI.Commands.RequestBoxType1 AND NOT gHMI.Commands.LoadRecipeType1;
_p13 := gHMI.Commands.RequestBoxType1;
IF _p12 THEN
    gHMI.StatusDatapoints.RecipeDialogSDP.0 := FALSE;
    gHMI.Commands.RequestBoxType2 := FALSE;
END_IF;
_p14 := _p13 AND gHMI.Commands.CancelBoxChange;
IF _p13 AND gHMI.Commands.CancelBoxChange THEN gHMI.Commands.RequestBoxType1 := FALSE; END_IF;
IF _p14 THEN
    gHMI.Commands.CancelBoxChange := FALSE;
    gHMI.StatusDatapoints.RecipeDialogSDP.0 := TRUE;
END_IF;
_p15 := _p13 AND gHMI.Commands.ConfirmBoxChange;
IF _p13 AND gHMI.Commands.ConfirmBoxChange THEN gHMI.Commands.LoadRecipeType1 := TRUE; END_IF;
IF _p15 THEN
    gHMI.Commands.ConfirmBoxChange := FALSE;
    gHMI.Commands.RequestBoxType1 := FALSE;
    gHMI.StatusDatapoints.RecipeDialogSDP.0 := TRUE;
END_IF;

(* Network 36 *)
_p16 := gHMI.Commands.RequestBoxType2 AND NOT gHMI.Commands.LoadRecipeType2;
_p17 := gHMI.Commands.RequestBoxType2;
IF _p16 THEN
    gHMI.StatusDatapoints.RecipeDialogSDP.0 := FALSE;
    gHMI.Commands.RequestBoxType1 := FALSE;
END_IF;
_p18 := _p17 AND gHMI.Commands.CancelBoxChange;
IF _p17 AND gHMI.Commands.CancelBoxChange THEN gHMI.Commands.RequestBoxType2 := FALSE; END_IF;
IF _p18 THEN
    gHMI.Commands.CancelBoxChange := FALSE;
    gHMI.StatusDatapoints.RecipeDialogSDP.0 := TRUE;
END_IF;
_p19 := _p17 AND gHMI.Commands.ConfirmBoxChange;
IF _p17 AND gHMI.Commands.ConfirmBoxChange THEN gHMI.Commands.LoadRecipeType2 := TRUE; END_IF;
IF _p19 THEN
    gHMI.Commands.ConfirmBoxChange := FALSE;
    gHMI.Commands.RequestBoxType2 := FALSE;
    gHMI.StatusDatapoints.RecipeDialogSDP.0 := TRUE;
END_IF;

(* Network 37 *)
_e20(CLK := gHMI.Commands.LoadRecipeType1);
IF _e20.Q THEN
    gRecipeInterface.Commands.LoadRecipe := TRUE;
    gHMI.Commands.LoadRecipeType2 := FALSE;
    gHMI.StatusDatapoints.RecipeReq2SDP.1 := FALSE;
    gHMI.StatusDatapoints.RecipeReq1SDP.1 := TRUE;
    gRecipeInterface.Parameters.RecipeName := TYPE1_RECIPE_NAME;
END_IF;

(* Network 38 *)
_e21(CLK := gHMI.Commands.LoadRecipeType2);
IF _e21.Q THEN
    gRecipeInterface.Commands.LoadRecipe := TRUE;
    gHMI.Commands.LoadRecipeType1 := FALSE;
    gHMI.StatusDatapoints.RecipeReq2SDP.1 := TRUE;
    gHMI.StatusDatapoints.RecipeReq1SDP.1 := FALSE;
    gRecipeInterface.Parameters.RecipeName := TYPE2_RECIPE_NAME;
END_IF;

(* Network 39 *)
gHMI.StatusDatapoints.RecipeIndexSDP := gRecipeInterface.Status.LoadedRecipeIndex;

(* Network 40 *)
_p22 := NOT gHMI.Commands.LoadRecipeType1 AND NOT gHMI.Commands.LoadRecipeType2;
IF _p22 THEN gHMI.Commands.LoadRecipeType1 := gHMI.StatusDatapoints.RecipeIndexSDP = 1; END_IF;

(* Network 41 *)
_p23 := NOT gHMI.Commands.LoadRecipeType1 AND NOT gHMI.Commands.LoadRecipeType2;
IF _p23 THEN gHMI.Commands.LoadRecipeType2 := gHMI.StatusDatapoints.RecipeIndexSDP = 2; END_IF;

(* Network 42 *)
IF gRecipeInterface.Status.Busy THEN gHMI.ColorMapDatapoints.RecipeSystemBusy := OK; END_IF;

(* Network 43 *)
IF NOT gRecipeInterface.Status.Busy THEN gHMI.ColorMapDatapoints.RecipeSystemBusy := NOTOK; END_IF;

(* Network 44 *)
SettingsLoaded := gRecipeInterface.Parameters.RecipeName = gRecipeInterface.Status.LoadedRecipeName;

(* Network 45 *)
IF SettingsLoaded THEN gHMI.ColorMapDatapoints.RecipeLoaded := OK; END_IF;

(* Network 46 *)
IF SettingsLoaded THEN gHMI.ColorMapDatapoints.RecipeLoaded := OK; END_IF;

(* Network 47 *)
IF NOT gAlarmActive THEN gHMI.BitmapSelectDatapoints.AlarmActive := ALARM_INACTIVE; END_IF;

(* Network 48 *)
IF gAlarmActive THEN gHMI.BitmapSelectDatapoints.AlarmActive := ALARM_ACTIVE; END_IF;

(* Network 49 *)
IF NOT gAdhesiveCtrlInterface.Status.AlarmActive THEN
    gHMI.ColorMapDatapoints.AdhesiveSystemOK := OK;
END_IF;

(* Network 50 *)
IF gAdhesiveCtrlInterface.Status.AlarmActive THEN
    gHMI.ColorMapDatapoints.AdhesiveSystemOK := NOTOK;
END_IF;

(* Network 51 *)
IF NOT gAirPressureAlarmActive THEN gHMI.ColorMapDatapoints.AirPressureOK := OK; END_IF;

(* Network 52 *)
IF gAirPressureAlarmActive THEN gHMI.ColorMapDatapoints.AirPressureOK := NOTOK; END_IF;

(* Network 53 *)
IF NOT gVacCtrlInterface.Status.AlarmActive THEN gHMI.ColorMapDatapoints.VacuumOK := OK; END_IF;

(* Network 54 *)
IF gVacCtrlInterface.Status.AlarmActive THEN gHMI.ColorMapDatapoints.VacuumOK := NOTOK; END_IF;

(* Network 55 *)
IF NOT gSafetyNotOKAlarmActive THEN gHMI.ColorMapDatapoints.SafetyOK := OK; END_IF;

(* Network 56 *)
IF gSafetyNotOKAlarmActive THEN gHMI.ColorMapDatapoints.SafetyOK := NOTOK; END_IF;

(* Network 57 *)
IF NOT gServoFeedInterface.Status.Error AND NOT gBodyHopperInterface.Status.Error AND NOT gLeftHopperInterface.Status.Error AND NOT gRightHopperInterface.Status.Error AND NOT gServoRamInterface.Status.Error AND NOT gFoldPushCtrlInterface.Parameters.LinMotBotFolder.Status.Error AND NOT gFoldPushCtrlInterface.Parameters.LinMotTopFolder.Status.Error THEN
    gHMI.ColorMapDatapoints.DriveFaultOK := OK;
END_IF;

(* Network 58 *)
IF gServoFeedInterface.Status.Error OR gBodyHopperInterface.Status.Error OR gLeftHopperInterface.Status.Error OR gRightHopperInterface.Status.Error OR gServoRamInterface.Status.Error OR gFoldPushCtrlInterface.Parameters.LinMotBotFolder.Status.Error OR gFoldPushCtrlInterface.Parameters.LinMotTopFolder.Status.Error THEN
    gHMI.ColorMapDatapoints.DriveFaultOK := NOTOK;
END_IF;

(* Network 59 *)
IF gIO.DIs.DownstreamSensor THEN gHMI.ColorMapDatapoints.DownstreamSensorOK := NOTOK; END_IF;

(* Network 60 *)
IF NOT gIO.DIs.DownstreamSensor THEN gHMI.ColorMapDatapoints.DownstreamSensorOK := OK; END_IF;

(* Network 61 *)
IF NOT gFoldPushCtrlInterface.Status.TopFoldValveStatus THEN
    gHMI.ColorMapDatapoints.Valve1OK := NOTOK;
END_IF;

(* Network 62 *)
IF gFoldPushCtrlInterface.Status.TopFoldValveStatus THEN gHMI.ColorMapDatapoints.Valve1OK := OK; END_IF;

(* Network 63 *)
IF NOT gFoldPushCtrlInterface.Status.BottomFoldValveStatus THEN
    gHMI.ColorMapDatapoints.Valve2OK := NOTOK;
END_IF;

(* Network 64 *)
IF gFoldPushCtrlInterface.Status.BottomFoldValveStatus THEN
    gHMI.ColorMapDatapoints.Valve2OK := OK;
END_IF;

(* Network 65 *)
IF NOT gFoldPushCtrlInterface.Status.CompOnValveStatus THEN
    gHMI.ColorMapDatapoints.Valve3OK := NOTOK;
END_IF;

(* Network 66 *)
IF gFoldPushCtrlInterface.Status.CompOnValveStatus THEN gHMI.ColorMapDatapoints.Valve3OK := OK; END_IF;

(* Network 67 *)
IF NOT gFoldPushCtrlInterface.Status.PushValveStatus THEN
    gHMI.ColorMapDatapoints.Valve4OK := NOTOK;
END_IF;

(* Network 68 *)
IF gFoldPushCtrlInterface.Status.PushValveStatus THEN gHMI.ColorMapDatapoints.Valve4OK := OK; END_IF;

(* Network 69 *)
IF gFoldPushCtrlInterface.Status.HardwireConfig THEN
    gHMI.StatusDatapoints.HardwireValveSDP := UNHIDE + UNLOCK;
END_IF;

(* Network 70 *)
IF gIO.SafetyStatus.SafetyProgramRunning THEN gHMI.StatusDatapoints.SafetyStartingSDP := HIDE; END_IF;

(* Network 71 *)
IF NOT gIO.SafetyStatus.SafetyProgramRunning THEN
    gHMI.StatusDatapoints.SafetyStartingSDP := UNHIDE;
END_IF;

(* Network 72 *)
_e24(CLK := gAlarmActive);
IF _e24.Q THEN gChangePage := PAGE_ALARM; END_IF;

(* Network 73 *)
IF gModeControlInterface.Parameters.MachineType = MACHINE_TYPE_BLISS THEN
    gHMI.StatusDatapoints.BlissSDP := UNHIDE + UNLOCK;
END_IF;

(* Network 74 *)
IF gModeControlInterface.Parameters.MachineType <> MACHINE_TYPE_BLISS THEN
    gHMI.StatusDatapoints.BlissSDP := HIDE + LOCK;
END_IF;

(* Network 75 *)
_t25 := gModeControlInterface.Parameters.MachineType = MACHINE_TYPE_CLASSICPAK;
IF _t25 THEN
    gModeControlInterface.Parameters.MaxPPM := 20;
    gModeControlInterface.Parameters.MinPPM := 0;
END_IF;

(* Network 76 *)
_t26 := gModeControlInterface.Parameters.MachineType = MACHINE_TYPE_BLISS;
IF _t26 THEN
    gModeControlInterface.Parameters.MaxPPM := 25;
    gModeControlInterface.Parameters.MinPPM := 0;
END_IF;

(* Network 77 *)
_t27 := gModeControlInterface.Parameters.MachineType = MACHINE_TYPE_TRAY;
IF _t27 THEN
    gModeControlInterface.Parameters.MaxPPM := 25;
    gModeControlInterface.Parameters.MinPPM := 0;
    gHMI.StatusDatapoints.TraySDP := UNHIDE + UNLOCK;
END_IF;

(* Network 78 *)
IF gModeControlInterface.Parameters.MachineType <> MACHINE_TYPE_TRAY THEN
    gHMI.StatusDatapoints.TraySDP := HIDE + LOCK;
END_IF;

(* Network 79 *)
_p28 := gModeControlInterface.Parameters.MaxPPM < gModeControlInterface.Parameters.PiecesPerMinute;
IF _p28 THEN
    gModeControlInterface.Parameters.PiecesPerMinute := gModeControlInterface.Parameters.MaxPPM;
END_IF;

(* Network 80 *)
_p29 := gModeControlInterface.Parameters.MinPPM > gModeControlInterface.Parameters.PiecesPerMinute;
IF _p29 THEN
    gModeControlInterface.Parameters.PiecesPerMinute := gModeControlInterface.Parameters.MinPPM;
END_IF;

(* Network 81 *)
LogoutTimer(IN := NOT ResetTimeoutTimer, PT := T#300s);
ResetUserLevel := LogoutTimer.Q;

(* Network 82 *)
_e30(CLK := ResetUserLevel);
IF _e30.Q THEN
    gUserLevel := 0;
    gChangePage := 0;
END_IF;

(* Network 83 *)
ResetTimeoutTimer := gActivePage <> OldPage;

(* Network 84 *)
OldPage := gActivePage;

(* Network 85 *)
gHMI.StatusDatapoints.LinMotSDP.0 := NOT gFoldPushCtrlInterface.Status.LinMotConfig;
gHMI.StatusDatapoints.LinMotTopHomeSDP.0 := NOT gFoldPushCtrlInterface.Status.LinMotConfig;
gHMI.StatusDatapoints.LinMotBotHomeSDP.0 := NOT gFoldPushCtrlInterface.Status.LinMotConfig;

(* Network 86 *)
_p31 := gHMI.ColorMapDatapoints.AutoModeSelected.0;
gHMI.StatusDatapoints.LinMotTopHomeSDP.1 := gHMI.ColorMapDatapoints.AutoModeSelected.0;
gHMI.StatusDatapoints.LinMotBotHomeSDP.1 := _p31;

(* Network 87 *)
gHMI.StatusDatapoints.PnuematicFolderSDP.0 := NOT gFoldPushCtrlInterface.Status.PneumaticConfig;

(* Network 88 *)
IF gAdhesiveCtrlInterface.Status.ATS_AddOnOverLimit THEN
    gHMI.ColorMapDatapoints.ATSAddOnOver := NOTOK;
END_IF;

(* Network 89 *)
IF NOT gAdhesiveCtrlInterface.Status.ATS_AddOnOverLimit THEN
    gHMI.ColorMapDatapoints.ATSAddOnOver := OK;
END_IF;

(* Network 90 *)
IF gAdhesiveCtrlInterface.Status.ATS_AddOnUnderLimit THEN
    gHMI.ColorMapDatapoints.ATSAddOnUnder := NOTOK;
END_IF;

(* Network 91 *)
IF NOT gAdhesiveCtrlInterface.Status.ATS_AddOnUnderLimit THEN
    gHMI.ColorMapDatapoints.ATSAddOnUnder := OK;
END_IF;

(* Network 92 *)
gAdhesiveCtrlInterface.Parameters.NordsonComms.ChannelDataSize := SIZEOF(in := gAdhesiveCtrlInterface.Parameters.NordsonComms.ChannelSetTempActual);

(* Network 93: Flash save set temp button if  requested temps are different from current set temps *)
gAdhesiveCtrlInterface.Parameters.NordsonComms.ChannelDataCmpResult := brsmemcmp(pMem1 := ADR(gAdhesiveCtrlInterface.Parameters.NordsonComms.ChannelSetTempActual), pMem2 := ADR(gAdhesiveCtrlInterface.Parameters.NordsonComms.ChannelSetTempRequested), length := gAdhesiveCtrlInterface.Parameters.NordsonComms.ChannelDataSize);

(* Network 94 *)
gHMI.ColorMapDatapoints.NordsonEditTemps := gAdhesiveCtrlInterface.Parameters.NordsonComms.ChannelDataCmpResult <> 0;

(* Network 95 *)
gHMI.ColorMapDatapoints.NordsonEditTemps.0 := gHMI.ColorMapDatapoints.NordsonEditTemps.0 AND FlashON.Q;

(* Network 96 *)
IF gIO.DIs.BodyHopperLow OR gIO.DIs.LeftHopperLow OR gIO.DIs.RightHopperLow THEN
    gHMI.StatusDatapoints.HopperLowSDP := UNHIDE + UNLOCK;
END_IF;

(* Network 97 *)
IF NOT gIO.DIs.BodyHopperLow OR NOT gIO.DIs.LeftHopperLow OR NOT gIO.DIs.RightHopperLow THEN
    gHMI.StatusDatapoints.HopperLowSDP := HIDE + LOCK;
END_IF;

(* Network 98 *)
_p32 := NOT gHMI.Commands.CycleServoRam;
IF _p32 THEN gHMI.StatusDatapoints.HomeServoRamSDP := UNHIDE + UNLOCK; END_IF;

(* Network 99 *)
_p33 := gHMI.Commands.CycleServoRam;
IF _p33 THEN gHMI.StatusDatapoints.HomeServoRamSDP := HIDE + LOCK; END_IF;

(* Network 100 *)
IF LubricationOK THEN gHMI.StatusDatapoints.LubeSDP := HIDE + LOCK; END_IF;

(* Network 101 *)
IF NOT LubricationOK THEN gHMI.StatusDatapoints.LubeSDP := UNHIDE + UNLOCK; END_IF;

(* Network 102 *)
_e34(CLK := gHMI.StatusDatapoints.AdhesivePatternConfirmedSDP.0);
IF _e34.Q THEN
    gHMI.StatusDatapoints.AdhesivePatternConfirmDialogSDP.0 := TRUE;
    gHMI.StatusDatapoints.AdhesivePatternDialogSDP.0 := TRUE;
END_IF;

(* Network 103: Controls whether or not the text is shown on screen for the respective hopper switches being off. Setting the first bit true hides the text *)
gHMI.StatusDatapoints.BodyHopperSwitchSDP.0 := gIO.DIs.BodyHopperMotor_RUN;

(* Network 104 *)
gHMI.StatusDatapoints.LeftHopperSwitchSDP.0 := gIO.DIs.LeftHopperMotor_RUN;

(* Network 105 *)
gHMI.StatusDatapoints.RightHopperSwitchSDP.0 := gIO.DIs.RightHopperMotor_RUN;
END_PROGRAM
```

### Program Logical/Libraries/AxisFUBs

#### AxisHandler.c
```c
#include <bur/plctypes.h>
#include "string.h"

#ifdef __cplusplus
	extern "C"
	{
#endif
#include "AxisFUBs.h"
#ifdef __cplusplus
	};
#endif
/* Implements state machine for single axis handling */
void AxisHandler(struct AxisHandler* t)
{

	if(t->AlarmActive == 1) {
		t->state = AXIS_STATE_ERROR;
	}

	//force these off. State machine will set them if jog is requested and state allows it
	t->pInterface->Commands.ToMapp.JogNeg = 0;
	t->pInterface->Commands.ToMapp.JogPos = 0;
	t->pInterface->Parameters.MovementParameters.Deceleration = t->pInterface->Parameters.MovementParameters.Acceleration;

	t->pInterface->Parameters.MovementParameters.Jog.LowerLimit = 0;

	t->DriveReadyTimeout.IN = 0; //will be set true in appropriate state(s)

	//	switch (t->axisInitState){
	//		//init the axis/drive
	//		case AXIS_INIT_TRANSFER_PARS:
	//
	//		//	strcpy((char*)&t->pInterface->Status.AxisState, "Loading Axis Parameters");
	//
	//		//	if(t->pSystemInterface->Status.DefaultRecipeLoaded == 1) //axis parameters should be part of the recipe system and are only 'good' once recipe system has loaded the values
	//			if(1)
	//			{
	//				//unclear if axis parameters will become part of the recipe system, so just continue on for now - jdl
	////				t->pInterface->Commands.ToMapp.SaveConfig = 1;
	////
	////				if(t->pInterface->Status.ConfigCommandDone){
	////					t->pInterface->Commands.ToMapp.SaveConfig = 0;
	////				}
	//
	//				t->axisInitState = AXIS_INIT_RETRIEVE_PARS;
	//			}
	//			break;
	//
	//		//Get mapp config parameters. These should ideally come from the recipe system
	//		case AXIS_INIT_RETRIEVE_PARS:
	//
	//		//	strcpy((char*)&t->pInterface->Status.AxisState, "Retrieving Axis Parameters");
	//
	//			t->pInterface->Commands.ToMapp.LoadConfig = 1;
	//
	//			if(t->pInterface->Status.ConfigCommandDone){
	//				t->pInterface->Commands.ToMapp.LoadConfig = 0;
	//				t->axisInitState = AXIS_INIT_WAIT_FOR_INIT;
	//			}
	//			break;
	//
	//		//Get mapp config parameters. These should ideally come from the recipe system
	//		case AXIS_INIT_WAIT_FOR_INIT:
	//
	//			//	strcpy((char*)&t->pInterface->Status.AxisState, "Retrieving Axis Parameters");
	//
	//			t->pInterface->Commands.ToMapp.Update = 1;
	//
	//			if(t->pInterface->Status.AxisInitialized){
	//				t->axisInitState = AXIS_INIT_DONE;
	//			}
	//			break;
	//
	//		case AXIS_INIT_DONE:
	//			if(t->pInterface->Commands.Init){
	//				t->pInterface->Commands.Init = 0;
	//				t->axisInitState = AXIS_INIT_TRANSFER_PARS;
	//			}
	//	}

	switch (t->state)
	{
		case AXIS_STATE_INIT:

			if (t->pInterface->Status.AxisBasicActive) {

				//force parameter save to the drive. values are set in init code of motion handler
				t->pInterface->Commands.ToMapp.SaveConfig = 1;

				if(t->pInterface->Status.ConfigCommandDone){
					t->pInterface->Commands.ToMapp.SaveConfig = 0;
					t->pInterface->Commands.ToMapp.Update = 0;
				}
				t->state = AXIS_STATE_POWERON_PREP;
			}
			break;

		//we need at least one scan where the power on command is 0. handles cases where the power on command is always true and the machine can't power on.
		case AXIS_STATE_POWERON_PREP:

			t->pInterface->Commands.ToMapp.Update = 1;

			if (t->pInterface->Status.AxisInitialized) {
				t->pInterface->Commands.ToMapp.Power = 0;
				t->state = AXIS_STATE_POWERON;
			}
			break;

		//power on the Drive
		case AXIS_STATE_POWERON:

			strcpy((char*)&t->pInterface->Status.AxisState, "Powering On");
			t->DriveReadyTimeout.IN = 1; //will be cleared outside of state machine

			if ((t->pInterface->Status.ReadyToPowerOn) || (t->DriveReadyTimeout.Q))  //Issue the power on command if drives do not become ready with in time out.  The drive will then post an alarm to explain why it won't power on.
			{
				t->DriveReadyTimeout.IN = 0;
				t->pInterface->Commands.ToMapp.Power = 1;

				if(t->pInterface->Status.PoweredOn)
				{
					t->state = AXIS_STATE_HOME;
				}
			}
			break;

		//On start up, home the axis
		case AXIS_STATE_HOME:

			strcpy((char*)&t->pInterface->Status.AxisState, "Waiting To Start Home");

			if(t->pInterface->Status.ReadyToPowerOn == 1)
			{
				if((*(t->FirstHomeExecuted) == 0) || (!t->pInterface->Status.Homed))
				{
					//if system is simulated or the home mode is direct home, just direct home
					if((t->IsSimulated) || (t->pHomingParameters->Mode == mpAXIS_HOME_MODE_DIRECT)) {
					//if(t->IsSimulated) {
					t->pInterface->Parameters.MovementParameters.Home.Position = 0;
					t->pInterface->Parameters.MovementParameters.Home.SensorOffset = 0;
					t->pInterface->Parameters.MovementParameters.Home.Mode = mpAXIS_HOME_MODE_DIRECT;

					t->pInterface->Commands.RequestHome = 0;
					t->pInterface->Commands.ToMapp.Home = 1;
					t->state = AXIS_STATE_W_HOME;
					}
					else if(t->pInterface->Commands.RequestHome) //Otherwise execute set home routine
					{
					memcpy(&t->pInterface->Parameters.MovementParameters.Home, t->pHomingParameters, sizeof(t->pInterface->Parameters.MovementParameters.Home));

					t->pInterface->Commands.RequestHome = 0;
					t->pInterface->Commands.ToMapp.Home = 1;
					t->state = AXIS_STATE_W_HOME;
					}
				}
					//				else if(!t->pInterface->Status.Homed) //got to this state with a good stored position but we aren't homed, so recall the position
					//				{
					//					t->pInterface->Parameters.MovementParameters.Home.SensorOffset = 0;
					//					t->pInterface->Parameters.MovementParameters.Home.Mode = mpAXIS_HOME_MODE_RESTORE_POS;
					//					t->pInterface->Commands.ToMapp.Home = 1;
					//					t->state = AXIS_STATE_W_HOME;
					//				}
				else if(t->pInterface->Status.Homed) //got to this state without requesting home, and we're already homed. Probably recovering from error, just go to idle
				{
					t->state = AXIS_STATE_IDLE;
				}
			}
			break;

		// wait for home to finish
		case AXIS_STATE_W_HOME:

			strcpy((char*)&t->pInterface->Status.AxisState, "Homing");

			if(t->pInterface->Status.Homed)
			{
				t->pInterface->Commands.ToMapp.Home = 0;
				*(t->FirstHomeExecuted) = 1; //a home has been completed successfully, we do not need the home routine again
				t->state = AXIS_STATE_IDLE;
			}
			break;

		//Idle state. Ready to receive commands for commands
		case AXIS_STATE_IDLE:

			strcpy((char*)&t->pInterface->Status.AxisState, "Idle");

			t->pInterface->Commands.StopPowerSaver = 0;

			if(t->pInterface->Commands.RequestHome == 1)
			{
				*t->FirstHomeExecuted = 0;
				t->state = AXIS_STATE_HOME;
			}
			else if(t->pInterface->Commands.RequestMoveAbs == 1)
			{
				t->pInterface->Commands.RequestMoveAbs = 0;
				t->pInterface->Commands.ToMapp.MoveAbs = 1;
				t->state = AXIS_STATE_MOVE;
			}
			else if(t->pInterface->Commands.RequestMoveAdditive == 1)
			{
				t->pInterface->Commands.RequestMoveAdditive = 0;
				t->pInterface->Commands.ToMapp.MoveAdditive = 1;
				t->state = AXIS_STATE_MOVE;
			}
			else if(t->pInterface->Commands.RequestMoveVelocity == 1)
			{
				t->pInterface->Commands.ToMapp.MoveVelocity = 1;
				t->state = AXIS_STATE_MOVE_VELOCITY;
			}
			else if(t->pInterface->Commands.RequestJogNeg)
			{
				t->pInterface->Commands.ToMapp.JogNeg = 1;
			}
			else if(t->pInterface->Commands.RequestJogPos)
			{
				t->pInterface->Commands.ToMapp.JogPos = 1;
			}
			else if(t->pInterface->Commands.RequestCoupleToMaster)
			{
				t->pInterface->Commands.ToMapp.CoupleToMaster = 1;
				t->state = AXIS_STATE_W_COUPLE;
			}

			///////////////////////////////////////////////////////////////////////////////////////////////////

			else if (t->pInterface->Commands.StartPowerSaver == 1)
			{
				// if power is removed in the program, wait in power saver mode
				t->pInterface->Commands.StartPowerSaver = 0;
				t->pInterface->Status.PowerSaverModeOn = 1;
				t->pInterface->Commands.ToMapp.Power = 0;
				t->state = AXIS_STATE_POWERSAVER;
			}
			break;

		case AXIS_STATE_POWERSAVER:

			t->pInterface->Commands.StartPowerSaver = 0;
			if (t->pInterface->Commands.StopPowerSaver == 1)
			{
				// if power is restored, wait for power to come back
				t->pInterface->Commands.StopPowerSaver = 0;
				t->pInterface->Commands.ToMapp.Power = 1;
				t->state = AXIS_STATE_POWERBACK;
			}
			break;

		case AXIS_STATE_POWERBACK:

			t->pInterface->Commands.StartPowerSaver = 0;
			t->pInterface->Commands.StopPowerSaver = 0;
			if(t->pInterface->Status.PoweredOn)
			{
				// when power is back, go to idle
				t->pInterface->Status.PowerSaverModeOn = 0;
				t->state = AXIS_STATE_IDLE;
			}
			///////////////////////////////////////////////////////////////////////////////////////////////////

		case AXIS_STATE_MOVE:

			strcpy((char*)&t->pInterface->Status.AxisState, "In Motion");

			if((t->pInterface->Status.InPosition == 1) && (t->pInterface->Status.MappCommandBusy == 0)){
				t->pInterface->Status.MoveComplete = 1;
				t->pInterface->Commands.ToMapp.MoveAbs = 0;
				t->pInterface->Commands.ToMapp.MoveAdditive = 0;
				t->state = AXIS_STATE_IDLE;
			}
			break;

		case AXIS_STATE_MOVE_VELOCITY:

			strcpy((char*)&t->pInterface->Status.AxisState, "In Velocity");

			if(t->pInterface->Commands.RequestMoveVelocity == 0){
				t->pInterface->Commands.ToMapp.MoveVelocity = 0;
				t->state = AXIS_STATE_IDLE;
			}

			break;

		case AXIS_STATE_W_COUPLE:

			strcpy((char*)&t->pInterface->Status.AxisState, "Waiting To Couple To Master");

			if(t->pInterface->Status.InSync){
				t->state = AXIS_STATE_COUPLED;
			}

			break;

		case AXIS_STATE_COUPLED:

			strcpy((char*)&t->pInterface->Status.AxisState, "Coupled To Master");

			if(!(t->pInterface->Commands.RequestCoupleToMaster)){
				t->pInterface->Commands.ToMapp.CoupleToMaster = 0;

				if(!(t->pInterface->Status.InSync)){
					t->state = AXIS_STATE_IDLE;
				}
			}
			break;

		//Error state. handle errors and return to idle when errors are no longer present
		case AXIS_STATE_ERROR:

			strcpy((char*)&t->pInterface->Status.AxisState, "Machine In Error");

			t->pInterface->Commands.ToMapp.Home = 0;
			t->pInterface->Commands.Init = 0;
			t->pInterface->Commands.RequestJogNeg = 0;
			t->pInterface->Commands.RequestJogPos = 0;
			t->pInterface->Commands.RequestMoveAbs = 0;
			t->pInterface->Commands.RequestMoveAdditive = 0;
			t->pInterface->Commands.RequestHome = 0;
			t->pInterface->Commands.RequestCoupleToMaster = 0;
			t->pInterface->Commands.RequestMoveVelocity = 0;
			t->pInterface->Commands.ToMapp.JogNeg = 0;
			t->pInterface->Commands.ToMapp.JogPos = 0;
			t->pInterface->Commands.ToMapp.Home = 0;
			t->pInterface->Commands.ToMapp.MoveAbs = 0;
			t->pInterface->Commands.ToMapp.MoveVelocity = 0;
			t->pInterface->Commands.ToMapp.MoveAdditive = 0;
			t->pInterface->Commands.MoveVelocityTrigStop = 0;
			t->pInterface->Commands.ToMapp.CoupleToMaster = 0;
			t->pInterface->Commands.ToMapp.SaveConfig = 1;
			t->pInterface->Commands.StartPowerSaver = 0;
			t->pInterface->Commands.StopPowerSaver = 0;
			t->pInterface->Status.PowerSaverModeOn = 0;

			if(t->pInterface->Status.InMotion == 0){
				t->pInterface->Commands.ToMapp.Power = 0;
			}

			if(t->AlarmActive == 0)
			{
				//t->state = AXIS_STATE_INIT;
				t->state = 0; //go to whatever state 0 is for now. appropriate state should probably depend on how far we got through init process
			}

			break;
	}

	//handle drive time out because it will not become ready
	t->DriveReadyTimeout.PT = 20000;  //wait 20 seconds for drive to become ready before timing out.
	TON(&t->DriveReadyTimeout);
}
```

### Constants.var
```iecst
VAR CONSTANT
	COUNTS_PER_ENCODER_REV : UINT := 23040;
	DEFAULT_RECIPE_NAME : STRING[255] := 'settings.xml';
	HIDE : USINT := 1;
	LOCK : USINT := 2;
	MAX_NUM_GLUE_CHANNELS : USINT := 4;
	MAX_NUM_GLUE_CHANNELS_M1 : USINT := MAX_NUM_GLUE_CHANNELS-1;
	MAX_NUM_ONOFF_PATTERNS : USINT := 4;
	MAX_NUM_ONOFF_PATTERNS_M1 : USINT := MAX_NUM_ONOFF_PATTERNS-1;
	NOTOK : USINT := 0;
	OK : USINT := 1;
	PPM_TO_DEG_PER_S : REAL := 6.0;
	UNHIDE : USINT := 0;
	UNLOCK : USINT := 0;
	ALARM_INACTIVE : USINT := 0;
	ALARM_ACTIVE : USINT := 1;
	PAGE_ALARM : USINT := 100;
	PUMPS_OFF : USINT := 16#0;
	PUMPS_ON : USINT := 16#2;
	MELTER_OFF : USINT := 16#0;
	MELTER_ON : USINT := 16#1;
	STANDBY_ON : USINT := 16#40; (*bit 6 on*)
	WRITE_COMMAND : USINT := 16#6;
	READ_COMMAND : USINT := 16#3;
	TEMP_UNIT_IDX : USINT := 110;
	TEMP_UNIT_START_CHANNEL : USINT := 0;
	IDX_SET_TEMP : USINT := 115;
	CHANNEL_SET_TEMP_START : USINT := 1;
	IDX_MELTER_STATUS : USINT := 10;
	IDX_ATS_ALARMS : USINT := 229;
	IDX_ACT_TEMP : USINT := 120;
	CHANNEL_ACT_TEMP_START : USINT := 1;
	IDX_ADHESIVE_HOUR : USINT := 225;
	CHANNEL_ADHESIVE_HOUR : USINT := 0;
	MAX_NUM_TEMP_CHANNELS : USINT := 5;
	MAX_NUM_TEMP_CHANNELS_M1 : USINT := MAX_NUM_TEMP_CHANNELS-1;
	MACHINE_TYPE_BLISS : USINT := 3;
	MACHINE_TYPE_CLASSICPAK : USINT := 1;
	MACHINE_TYPE_TRAY : USINT := 2;
	NUM_NORDSON_TEMP_ZONES : USINT := 10;
	NUM_NORDSON_TEMP_ZONES_M1 : USINT := NUM_NORDSON_TEMP_ZONES-1;
	TYPE1_RECIPE_NAME : STRING[80] := 'settings1.xml';
	TYPE2_RECIPE_NAME : STRING[80] := 'settings2.xml';
	NUM_PNP_TRIES : USINT := 3;
	NUM_SIDE_TRIES : USINT := 3;
	NUM_FOLD_TRIES : USINT := 3;
END_VAR
```

### Library Logical/Libraries/MappCall

#### MappCall.fun
```iecst
{REDUND_ERROR} FUNCTION_BLOCK AxisBasic (*Implements config and basic for a mapp axis*) (*$GROUP=User,$CAT=User,$GROUPICON=User.png,$CATICON=User.png*)
	VAR_INPUT
		pMpLink : UDINT;
		pAxis : UDINT;
		pEndlessPosition : {REDUND_UNREPLICABLE} UDINT;
		AxisInterface : REFERENCE TO Axis_Interface_typ;
		OdometerValue : LREAL;
		Override : REAL;
		ErrorReset : BOOL;
	END_VAR
	VAR
		AxisBasic : {REDUND_UNREPLICABLE} MpAxisBasic;
		AxisConfig : MpAxisBasicConfig;
		AbsDistance : LREAL;
		zzInternalMemory : ARRAY[0..67] OF SINT; (*Internal memory*)
		SetOverride : MC_SetOverride;
	END_VAR
END_FUNCTION_BLOCK

FUNCTION StatusID_Decoder : USINT
	VAR_INPUT
		IN : MpAxisErrorEnum;
	END_VAR
END_FUNCTION

FUNCTION Severity_Decoder : UDINT
	VAR_INPUT
		IN : MpComSeveritiesEnum;
	END_VAR
END_FUNCTION

FUNCTION Facility_Decoder : UDINT
	VAR_INPUT
		EN : BOOL;
		IN : MpComFacilitiesEnum;
	END_VAR
END_FUNCTION
```

#### Severity_Decoder.st
```iecst
FUNCTION Severity_Decoder

	CASE IN OF

		mpCOM_SEV_SUCCESS:
			Severity_Decoder := 0;

		mpCOM_SEV_INFORMATIONAL:
			Severity_Decoder := 1;

		mpCOM_SEV_WARNING:
			Severity_Decoder := 2;

		mpCOM_SEV_ERROR:
			Severity_Decoder := 3;

	END_CASE

END_FUNCTION
```

#### StatusID_Decoder.st
```iecst
FUNCTION StatusID_Decoder

	CASE IN OF

		mpAXIS_NO_ERROR:
			StatusID_Decoder := 0;

		mpAXIS_ERR_ACTIVATION:
			StatusID_Decoder := 1;

		mpAXIS_ERR_MPLINK_NULL:
			StatusID_Decoder := 2;

		mpAXIS_ERR_MPLINK_INVALID:
			StatusID_Decoder := 3;

		mpAXIS_ERR_MPLINK_CHANGED:
			StatusID_Decoder := 4;

		mpAXIS_ERR_MPLINK_CORRUPT:
			StatusID_Decoder := 5;

		mpAXIS_ERR_MPLINK_IN_USE:
			StatusID_Decoder := 6;

		mpAXIS_ERR_PAR_NULL:
			StatusID_Decoder := 7;

		mpAXIS_ERR_CONFIG_NULL:
			StatusID_Decoder := 8;

		mpAXIS_ERR_CONFIG_NO_PV:
			StatusID_Decoder := 9;

		mpAXIS_ERR_CONFIG_LOAD:
			StatusID_Decoder := 10;

		mpAXIS_WRN_CONFIG_LOAD:
			StatusID_Decoder := 11;

		mpAXIS_ERR_CONFIG_SAVE:
			StatusID_Decoder := 12;

		mpAXIS_ERR_CONFIG_INVALID:
			StatusID_Decoder := 13;

		mpAXIS_ERR_AXIS_HANDLE_NULL:
			StatusID_Decoder := 14;

		mpAXIS_WRN_ERROR_TABLE_MISSING:
			StatusID_Decoder := 15;

		mpAXIS_WRN_CFG_WAIT_ERROR_RESET:
			StatusID_Decoder := 16;

		mpAXIS_WRN_CFG_WAIT_POWER_OFF:
			StatusID_Decoder := 17;

		mpAXIS_WRN_CFG_WAIT_STANDSTILL:
			StatusID_Decoder := 18;

		mpAXIS_ERR_PLC_OPEN:
			StatusID_Decoder := 19;

		mpAXIS_WRN_PLC_OPEN:
			StatusID_Decoder := 20;

		mpAXIS_WRN_READ_TORQUE_OFF:
			StatusID_Decoder := 21;

		mpAXIS_ERR_MAX_TORQUE_REACHED:
			StatusID_Decoder := 22;

		mpAXIS_ERR_SLAVE_NOT_FOUND:
			StatusID_Decoder := 23;

		mpAXIS_ERR_MASTER_NOT_FOUND:
			StatusID_Decoder := 24;

		mpAXIS_ERR_WRONG_DENOMINATOR:
			StatusID_Decoder := 25;

		mpAXIS_ERR_WRONG_NUMERATOR:
			StatusID_Decoder := 26;

		mpAXIS_ERR_NO_CAM_NAME:
			StatusID_Decoder := 27;

		mpAXIS_WRN_SLAVE_NOT_READY:
			StatusID_Decoder := 28;

		mpAXIS_ERR_CHECK_SLAVE_STATUS:
			StatusID_Decoder := 29;

		mpAXIS_ERR_CMD_WRONG_AXISTYPE:
			StatusID_Decoder := 30;

		mpAXIS_WRN_PARAMETER_LIMITED:
			StatusID_Decoder := 31;

		mpAXIS_WRN_MULTIPLE_COMMAND:
			StatusID_Decoder := 32;

		mpAXIS_ERR_CAM_PARAMETER:
			StatusID_Decoder := 33;

		mpAXIS_ERR_RECOVERY_NOT_ALLOWED:
			StatusID_Decoder := 34;

	END_CASE

END_FUNCTION
```

### Program Logical/Libraries/SetRamPars

#### ComputeDistanceMoved.st
```iecst
(* Compute how far encoder has moved *)
FUNCTION ComputeDistanceMoved

	IF((CurentPos -  OldPos) >= 0) THEN
		ComputeDistanceMoved := CurentPos -  OldPos;
	ELSE
		ComputeDistanceMoved := 711.2 + CurentPos -  OldPos;
	END_IF

END_FUNCTION
```
